(* CoDeSys 2.3 project: cy-01-wg-028.pro *)
(* Title: cy-001-wg (Albino Biblioteca E02) *)
(* Author: Andrea Ravasio *)
(* Libraries: Standard.lib 2.12.10 14:48:34, Util.lib 26.9.14 10:12:46, Visual.lib 2.12.10 14:48:34, LON_01.lib 28.9.12 14:05:10, WagoLibIdent.lib 25.2.13 11:12:16, WagoLibMBX_01.lib 20.3.12 16:32:40, WagoLibStatus.lib 2.12.10 14:48:32, SysLibFile.lib 2.12.10 14:48:34, SysLibRtc.lib 2.12.10 14:48:32, SysLibSockets.lib 10.2.11 09:20:54, SysLibEvent.lib 2.12.10 14:48:34, SysLibPlcCtrl.lib 2.12.10 14:48:32, SysLibCallback.lib 2.12.10 14:48:32 *)

(* PLC configuration (modules and I/O channels)
0750-1506 8DI / 8DO 24V DC 0.5A [Type_34_8_Channels] node 0, in %IB36 out %QB28 {INTTypePAAssignment = PLC; INTTypeModule = plugged}
  CIR09_AL AT %IX18.0 [BOOLOnX_I] Ch_1 Digital input
  CIR09_EN AT %QX14.0 [BOOLOnX_Q] Ch_1 Digital output
  CIR09_ST AT %IX18.1 [BOOLOnX_I] Ch_2 Digital input
  CIR08_EN AT %QX14.1 [BOOLOnX_Q] Ch_2 Digital output
  CIR02_ST AT %IX18.2 [BOOLOnX_I] Ch_3 Digital input
  CIR01_EN AT %QX14.2 [BOOLOnX_Q] Ch_3 Digital output
  CIR02_AL AT %IX18.3 [BOOLOnX_I] Ch_4 Digital input
  CIR01_ECO AT %QX14.3 [BOOLOnX_Q] Ch_4 Digital output
  CIR03_ST AT %IX18.4 [BOOLOnX_I] Ch_5 Digital input
  CIR07_EN AT %QX14.4 [BOOLOnX_Q] Ch_5 Digital output
  CIR03_AL AT %IX18.5 [BOOLOnX_I] Ch_6 Digital input
  CIR06_EN AT %QX14.5 [BOOLOnX_Q] Ch_6 Digital output
  CIR04_ST AT %IX18.6 [BOOLOnX_I] Ch_7 Digital input
  CIR05_EN AT %QX14.6 [BOOLOnX_Q] Ch_7 Digital output
  CIR04_AL AT %IX18.7 [BOOLOnX_I] Ch_8 Digital input
  CIR04_EN AT %QX14.7 [BOOLOnX_Q] Ch_8 Digital output
0750-1506 8DI / 8DO 24V DC 0.5A [Type_34_8_Channels] node 1, in %IB36 out %QB28 {INTTypePAAssignment = PLC; INTTypeModule = plugged}
  CIR05_ST AT %IX18.8 [BOOLOnX_I] Ch_1 Digital input
  CIR03_EN AT %QX14.8 [BOOLOnX_Q] Ch_1 Digital output
  CIR05_AL AT %IX18.9 [BOOLOnX_I] Ch_2 Digital input
  CIR02_EN AT %QX14.9 [BOOLOnX_Q] Ch_2 Digital output
  CIR06_ST AT %IX18.10 [BOOLOnX_I] Ch_3 Digital input
  AT %QX14.10 [BOOLOnX_Q] Ch_3 Digital output
  CIR06_AL AT %IX18.11 [BOOLOnX_I] Ch_4 Digital input
  AT %QX14.11 [BOOLOnX_Q] Ch_4 Digital output
  CIR07_ST AT %IX18.12 [BOOLOnX_I] Ch_5 Digital input
  AT %QX14.12 [BOOLOnX_Q] Ch_5 Digital output
  CIR07_AL AT %IX18.13 [BOOLOnX_I] Ch_6 Digital input
  AT %QX14.13 [BOOLOnX_Q] Ch_6 Digital output
  CIR01_ST AT %IX18.14 [BOOLOnX_I] Ch_7 Digital input
  AT %QX14.14 [BOOLOnX_Q] Ch_7 Digital output
  CIR01_AL AT %IX18.15 [BOOLOnX_I] Ch_8 Digital input
  AT %QX14.15 [BOOLOnX_Q] Ch_8 Digital output
0750-1506 8DI / 8DO 24V DC 0.5A [Type_34_8_Channels] node 2, in %IB37 out %QB29 {INTTypePAAssignment = PLC; INTTypeModule = plugged}
  CIR08_ST AT %IX19.0 [BOOLOnX_I] Ch_1 Digital input
  AT %QX15.0 [BOOLOnX_Q] Ch_1 Digital output
  CIR08_AL AT %IX19.1 [BOOLOnX_I] Ch_2 Digital input
  AT %QX15.1 [BOOLOnX_Q] Ch_2 Digital output
  ALARM_PM AT %IX19.2 [BOOLOnX_I] Ch_3 Digital input
  AT %QX15.2 [BOOLOnX_Q] Ch_3 Digital output
  ALARM_TB AT %IX19.3 [BOOLOnX_I] Ch_4 Digital input
  AT %QX15.3 [BOOLOnX_Q] Ch_4 Digital output
  ALARM_PB AT %IX19.4 [BOOLOnX_I] Ch_5 Digital input
  AT %QX15.4 [BOOLOnX_Q] Ch_5 Digital output
  CTL01_ST AT %IX19.5 [BOOLOnX_I] Ch_6 Digital input
  AT %QX15.5 [BOOLOnX_Q] Ch_6 Digital output
  AT %IX19.6 [BOOLOnX_I] Ch_7 Digital input
  AT %QX15.6 [BOOLOnX_Q] Ch_7 Digital output
  AT %IX19.7 [BOOLOnX_I] Ch_8 Digital input
  AT %QX15.7 [BOOLOnX_Q] Ch_8 Digital output
0750-1506 8DI / 8DO 24V DC 0.5A [Type_34_8_Channels] node 3, in %IB38 out %QB30 {INTTypePAAssignment = PLC; INTTypeModule = plugged}
  CIR01_TERM AT %IX19.8 [BOOLOnX_I] Ch_1 Digital input
  AT %QX15.8 [BOOLOnX_Q] Ch_1 Digital output
  CIR07_TERM AT %IX19.9 [BOOLOnX_I] Ch_2 Digital input
  AT %QX15.9 [BOOLOnX_Q] Ch_2 Digital output
  CIR05_TERM AT %IX19.10 [BOOLOnX_I] Ch_3 Digital input
  AT %QX15.10 [BOOLOnX_Q] Ch_3 Digital output
  CIR04_TERM AT %IX19.11 [BOOLOnX_I] Ch_4 Digital input
  AT %QX15.11 [BOOLOnX_Q] Ch_4 Digital output
  AT %IX19.12 [BOOLOnX_I] Ch_5 Digital input
  AT %QX15.12 [BOOLOnX_Q] Ch_5 Digital output
  AT %IX19.13 [BOOLOnX_I] Ch_6 Digital input
  AT %QX15.13 [BOOLOnX_Q] Ch_6 Digital output
  AT %IX19.14 [BOOLOnX_I] Ch_7 Digital input
  AT %QX15.14 [BOOLOnX_Q] Ch_7 Digital output
  AT %IX19.15 [BOOLOnX_I] Ch_8 Digital input
  AT %QX15.15 [BOOLOnX_Q] Ch_8 Digital output
0750-1506 8DI / 8DO 24V DC 0.5A [Type_34_8_Channels] node 4, in %IB39 out %QB31 {INTTypePAAssignment = PLC; INTTypeModule = plugged}
  KEY_CT_ST AT %IX20.0 [BOOLOnX_I] Ch_1 Digital input
  KEY_CT_EN AT %QX16.0 [BOOLOnX_Q] Ch_1 Digital output
  GZB_ST AT %IX20.1 [BOOLOnX_I] Ch_2 Digital input
  GZB_CTRL AT %QX16.1 [BOOLOnX_Q] Ch_2 Digital output
  VPN_ST1 AT %IX20.2 [BOOLOnX_I] Ch_3 Digital input
  VPN_DIS AT %QX16.2 [BOOLOnX_Q] Ch_3 Digital output
  VPN_ST2 AT %IX20.3 [BOOLOnX_I] Ch_4 Digital input
  VPN_CTRL1 AT %QX16.3 [BOOLOnX_Q] Ch_4 Digital output
  KEY_QE_ST AT %IX20.4 [BOOLOnX_I] Ch_5 Digital input
  VPN_CTRL2 AT %QX16.4 [BOOLOnX_Q] Ch_5 Digital output
  KEY_SCT_ST AT %IX20.5 [BOOLOnX_I] Ch_6 Digital input
  AT %QX16.5 [BOOLOnX_Q] Ch_6 Digital output
  AT %IX20.6 [BOOLOnX_I] Ch_7 Digital input
  TEST1 AT %QX16.6 [BOOLOnX_Q] Ch_7 Digital output
  AT %IX20.7 [BOOLOnX_I] Ch_8 Digital input
  TEST2 AT %QX16.7 [BOOLOnX_Q] Ch_8 Digital output
0750-0464#04 2/4 AI RTD / ADJ./ HA [Type_44_4_Channels] node 5, in %IB36 out %QB24 {INTTypePAAssignment = PLC; INTTypeModule = plugged}
  T_S01 AT %IW0 [INTOnW_I] Ch_1 signed Input value
  T_S05 AT %IW1 [INTOnW_I] Ch_2 signed Input value
  T_S03 AT %IW2 [INTOnW_I] Ch_3 signed Input value
  T_S04 AT %IW3 [INTOnW_I] Ch_4 signed Input value
0753-0648 LON-FTT [Type_55_1_Channels] node 6, in %IB36 out %QB24 {INTTypePAAssignment = PLC; INTTypeModule = plugged; DataStream = 1F8B0800000000000400ED5D796FDBC892FF7F81FD0E5C01FB9001AC5897E5631C3F2812150BA3C34349F6044920D0624BE68422F578D8F17EFAADEA2629526C5E3AE2D823609091C966755577F5AF8E2E362FFFFD63A1098FC4B45443FF5028BF2F1504A24F0D45D5E71F0A8E3D2B96EB857F5FFDF77F5D760DBDA3DBC49C; DataStream = C95322C043BA75F1C3523F141E6C7B79717CFCF4F4F4FEA9FADE30E7C79552A97CFC57AF3B9C3E90855C5475CB96F52929F84F29E94F15841BD3989BF2A2038DCF4B17A5D2C529FC7B72512A5F94EA17A51AFC28087FA9B3BEBC201F0A0DED5ED58D8958AA148421D1662D63EA2C886ECB3688D53416F81B5A298AF06C38A6; DataStream = 306557840762025B7DE29886DE56CDC5936C925B7F2CCE690743F991DCC8F6C38742F3E2EBD2B9BFD7D4A9F1B5A12B2691BFDEA9CBAF7F75DA05A167288E46FACEE29E98F06801464C1070CC7AB2F97D70FF3799DA16BDB67ED5BD08974764B1D4649B7414604D9DA9C4F4EFC15D1C8E8E72552A09BCFF2E8FDDFB81278653; DataStream = 6349AEE016FB11B8F30779C6EBF8BFC0D58EAE901F57E5CB63F6C3E7EB3881319F699C86AB61FB66A41B0A6192AD1EA437FD47B84DC34D06A63A577559E3360DDDF41FE9585D63FA9D2857B6E91090C1FB33D0A027EB8A6C1BE6B3DF667525D06CB044A591B5AB99AC59B4997FC56FD52338D16CBA7128437FFBAD448DA09A; DataStream = 350D07740D16CB85AE6A1F0AD87941380E0C08B19F0CF3FBAD6CAAF2BD46ACE0A4ACDD0BDC4AD398CDB42659737CED39AFACAB4F4085F066588752F588A34BFDDBD1C4B8FF7B6292FF38C48AD3A69546E98FAAE4358D3609294DB029579B3269540EADCAAE5951ED2AC768176D994DC31851551F125D19A90B3AB5C13FC3ED; DataStream = E41FA176813FD7DB49644AD44712681ABCB226FC8DA91AA66A3FAF84F7AF845A0E89F9A84EC9E81934AF31FDAE1B4F1A51E644016D0CDC093DD2524D400618C8AB8EBE7460525717C22C83599BA9539C9BABBEA10313C12BA1A64D439FA973C7A4060456C99298B64AACF541ED587E576BCAB27E3DF4D8C7679B0CD5FF2357; DataStream = D5CB63FF7760D51FC72FFB5F1611AA498850DD2522803B613B56064030866ECB543CF05BFEF2705039C04176381838F6EBC283FA9BC183D3243C38DD191ECC548DA08B90C53D68435B099BA6BB077ED31DE281AFE8E980E091CC800727073C78BBEE41B9F276F0A0968407B59DE241760701D7399AFE2C2EC2AAED2F0F0AF5; DataStream = 0328BC6127A172FA6650E13C92866223C4A286D24E5161696481046AFA6F8C2C41C3AAE92F0F08A7074078BB5E42DEA021726795714C65F9F29897BDDE2CA59D9CA02E966332D4C59C296ABA286F55D376644D9839FA94AD16E15E83415DCF3CE74A2327ACD5431E391BFEFF7A7964689E358F1CA59DC110F8DAB0434B9027; DataStream = 8114A765B4E5C11408BF9A6FE88B77C828B3117AB98C32B4CE98518E503E00C3DB028697F71173E2C2DBC92C9F256592CE769649B241B570F92E9659700115714832BA0C41D20760785BC0F0FA3C86B7934D3A3B4B4286B35D2183ACC9E6220B283458C32C90E0D23CA0C1DB428357E72654CE0F68B04F34C8EC231C00E14D; DataStream = 02C2EB730FDE1222246514CE769651C0989F64CA336ACF43D6360B22B8640F88F0B610E1F5B9086F060FCAA5241781DEDD0D223C3CCAD3C9C25032A142EBFA6E02939C3D9D10A07E0087B7050EAFCF5D28BF217438494487939D651AE1CA24539611A1A131B5B161C64CA34BFA800B6F0B170E4EC30116C2B000DEC28DA1EA; DataStream = 5977200EB8F02671E1F5F90B0760D83F301CFC857F3A2E1CFC85972B634A4285F39D8182F5A4DAD3872CA0D06CB71014441D472963EAD1257E8085B7050B0777E1800B215CF874C085032E1CDC85C39E843748619FA1479B1FF624FED1E0F0FA9C86C39EC41E730C080D8704C33F1D140E1EC3011322EEC26143E21F8F0BAF; DataStream = CF593800C3FE81E1E02FFCD371E1CDFB0BBB3E6463ED9A7575F93F5F9AADC6A8F1E532DB11DE974DD99635637E7589C7D6081D0BFE67139328785CB5D0829BAB93AF6B48039BE1147E28E0BFF0B7612E64DB6F54C7363DF96FC30C3C5710FCA3B2DDF3BB29194B78F7E3ACFEDB5710E10E86C4FA8A14ADAFC351A3DF6A48AD; DataStream = F7A3CF37ECC06F3CED3B06070B824466C0AF3E2589ADE89B98F86E25F053392E578F2BA57245289F5D544A17E54AE16A1DAD292BDCABC247D9724760082B756A7FA97F2B08740983F8058182E787C269B520202C7D28D08175CF82806B8F367B18710C241427C391346E8EFCA3CD6134D5297B3274966141402D43F60BC258; DataStream = 57A1B37F69F6EF1DFD51D65445B06C132616BAB10CC79C927FCDEDDFF94205D81775672178E491BB898D73F7435D380B2A0A800CFB5D2C7BC248F17288FD718F27852FFA509DEBAE62B9A27892CC024324E8F0945510903BC216833BA427088A29328D758BF6023A3587B9B0F070FA393B7C1DFE1A4EF1051AFAC74ACE9393; DataStream = EA89271EED8927DCB83FEC7CEA8BAD4977D0FF541006B399456C4A282AB0CA886067A41110B71212D76DB56F895C4817F0ED62C3E14E5C8C6C55FE645272139F5CBC940B55D3548B4C0D5DB132C90933FDA5BA5A4BFE026A81568095474D106445011DB7F8627406FD15FB273CF615D4729F0663F8C463D8C321BF938CEBBF; DataStream = B2E2B9E2F1DC6024041B1F03E0B5CDE7A4B59FC834B2637BDC563D6E793D64D5A5E1838114B32853B51AC0816A35221F3502093A35BC1E4869023222114DF2E1E1AC78AFDA82E3322F00E2310769BF2B273CC06A4E64A86F840CE57A9CA8EB8E0375A336B14FAE6971EE756217F10B0A496B2A937E5A7AFC52B238FDEC414B; DataStream = CB01252DBF261DFDA8DAFEE4AC09E4829FB190559DC7FEC7CEA89DA26F8AFB703CDBFE44B1A6B9AD92702A5011E09F804D74053A0D0A5439F544EA83326C28904E1F8D1787EA994E23AD3C42D42242D47C216A4121026615F05698629374514EF99694DA840459A818823113B0A94AB219D18D251A99B26EC934E4A1CE8299; DataStream = 2ED71977A1FC98B88FC78B461BC0E8C164E505F31CA050393909C35D1E1038E7229D4B265E32D622A8825B00F7E9B7E052622C7C320D67B93564CF97F1903D0FF5B03580A5A17058A536C2DE7BC3D088ACEF03B6EA2B15823E37E4DFA28F66006136F4ACF93FDE74303EC6BA6341DB994A346543511C4A224994B448FA604A; DataStream = 0EA62404C05B5B9239A3B29D4AF24DCB2606673397DB0578C77EC03D81298BD00D2EE2C40D4EB9C48D7881E4C448449FFC98BF896C5E8E3BAF54DCBCD01288E5906A0BC7A1F62DB842BD8C642D94916467506E9A90F49E76E3D7D3DDE724590FA19464B9CCCD490E6325894B49AEB84FCC48B266F109C9FAFE93107D1FB991; DataStream = A398BC57F6D424330413633671C9C5A7225C83B46F01874423539B5A782D394ACF909DB45C6213466C671958CC4C2664F936CD46CA8AE973B6B3ACBE0B013189D4A9A92E6D836B9033050E4A80C4AE396F98A6FCFCA55CFF86EADE6633343304192F0B846D95AE3C5EDC6AB1E82301BCF69FE209D890A4C6E714F928F43002; DataStream = 2E22D43DF1181FC05AB92E4C1F64131C1C62664812D3D5D1840732DA1E04D300CA55CE22C2AD0F09672ED992695E37A495C015AEADF525FE523EF9B6B666E2D09125BB1AC366A7B31A8ACD8D16EDE74F4756323A63E5DA69EDAC5AAF9DA6C566EE30FC396EB402C3C045464E8CB6267DCD37D2CF762E0F7A43641CA5A52DC3; DataStream = 8058C9133A675EB33B7544524133F3764860FBE67CB7F0C3D08785CE42A715833E5CF0F11FDA147C58203D51154FB628F6D405A67DFB8D7162C5DFD6B1F725FC12C19A6CD9F49F14DCD4D7464223FADC7ED83E0470E5F7C8C50F80D817CAB5F3D259B1ECA557BC677EB94C291624EC2655BAFB382E7DD321562AAE839977FF; DataStream = 214F84BE05CC96035B7CE5550DCA5935182211E1119CE364DF2F26E4A3870C72362BD185561F5505BFA1830B96AED31DE48C19BB48B1149F3A8AF20A0F94769333884F4CA6F05BCEC96F793FFC56B2F25BC9C96F653FFC56B3F25BCDC96F753FFCD6B2F25BCBC96F6D3FFC9E64E5F72427BF27FBE1B79E95DF7A4E7EEBFBE1; DataStream = F7342BBFA739F93DDD21BFD9383C4B4FD6735D1B78F6EC85C1F77C73D6CF5F1887CB09862E8DF7F29E8C5E66502E2758BD54E6F7640133237439C104A632BF27739819AECB09F63095F93DD9C6CCD85D4E308EA9CCEFC9506606F27282A54C653EB3D5DC59D59F1711F859182C8817E8D786368807569F2AF2B8F737809E89; DataStream = 6C1E090B43B71F8E04457E3E121E0C07AFA8BA63932381150467CC9A66CF9C554B58E5CFD91CFA4C647EC413CCA145C57CA68F25A5032B4189F3A40373C5AF9E183D1CD03CF12B37285F302AF1BA471BEC4998EA2A5126738BA1E344E146E28A9C58F100B7F72446C50FAAAF41B1F3C851E3C9F14089C40B82F7F724C9C9B9; DataStream = AF5D74716E5D23BB70C924E8176DB17779860C6472C8C32D1C72B12A29871578BD619BFC4D204F5E5EEDD89FF95B3FF42B319B6FD9D3CFC6F8C0B5978C79D770EB3F7224CCBD6712F2E5518134FFA197CD91C709BCE51AF2C4CB97204781B7CE8F6FB84FC55E3D8CD9F6C8F376844109B1ED8FD80D2BD628F3DE3DAD27A1EA; DataStream = 3FC1ADB0503949B512F218AAE1C566C76CBFB19A92C4BAB5557F499BA8B2DF4D7C85C9695611976EA1D244238F44CB5235E39736D127D225E596B185BB4D927619EA2E5EE2B39FF4921F0245FF364F3D0D77438BEAE1C4362688B3497AABAE3A15A6B26321D8BAB09C2A2FC3D91AC5D95B4CB1C7806C8D07B2B76CEF2C7547; DataStream = 92BF8DE3EEBCADED80FB505BFB2950CB9539C7560E1768A964B44C262114FBB9B0CA8298E4B8254E3BB988CA89625E41E852E682EAEB8C5DCA5CD87C85C10BBF78E895462FFC12A0571CBE54F87BF0B9E2975DA3D9F9796086FC57C1F354347103FF4590D6CEDE3E0F9A58E6FF69EA023CEC1C8636F0580673CB2FD7629EA3; DataStream = 4BE3658D6EC228E4D0CB04FF9892DECE006F117287CB795DE7F3DC37BFB4D67269586A5C7C9AA5481E9E8F44A94B3CFD8C98475E3DCFFE8B2325222BC777E07BA340B4F3D45249CE2B464F93A59D9211F535955657E3D4ADDE53DCFF3117BE90196AB5C238C3CDCB81C0B1555A3EC8ACDEAB5AD584EE5C277D47CA0DB4373F; DataStream = 4A0662E749E03496D071129DD6914FF9174A18FCC42C814B9877164EA5C60DA1D327241C42738D74B8DBA410DA0875171F4263A4BAA52206368F2AABDDA3F3EA9AE41B27245113C3AF10D5838AE8BE7833D3E4797633F766B431B558C3CDD9163B2D3A44E91B915CC55319153EEF3BD84A2D6713C253E71D48B25A433FBF94; DataStream = A3A55A4844D9460EC5A5F122E51C03C72E1AB322F5CAAC6DA4301C1B5F3063845EA4B863B0247A71AA9A5347DD4AAF0CA03371E9BC48A1873B27163B39710793E2527A91C28F1E993EC8BA0A1D1767B2A36D35330B9FD684D27A9162903621CABD3CFD0EE2A89A636E353F3397D6C4A5F593CAFE068FC42C9AB23ECFCA3C37; DataStream = 243780CA845279114B3206BBBA03291C24B34F31522C8888EFAE9AB9D7075716E2D3DAE7FA48B12863FACDA0A26D141744B6B22F9098D94162B8D3E2127B11CBD234160B47778F3AB0722E7CAE5C53A0B887459FDDC6B4A16FA2808DD166453BBB23C61506E59820A589BD373F2CADBCD093A3A8EAC5257288870F6D21932F; DataStream = CE44D5271EC117B137EC24E22298F26DE4D1289509FFF0CE7DD8989EAC3B80695343B74D43CBC83A3727B3A094262EA5178A5A96E093B1ADFB2D240155F26A727EBEA16132A0D13655252B78C589E19179110B2391A561DAC5856C7DDF460C939299209917B12A1E47AA3E2FE2D7B1B69165B9A245BFB4F52236252810DA84; DataStream = 5D0984B45EC4AAD0CD90A26ED8EAECB9A8E40BF5B952B12D104670B2DFB83FC5AA48C4E2BFEF9B69E1C03DC0E3C55223C93BA71B1CD17726044D8B5F0A897D9A8F44C9F0DA06778B2DF0FC3E4EDFDA22D1BF7A079B7E407383B4AAE53EB8967FA4A52E2CAB4AF6B26BB82A5B89AD365ADF218C2F357227C57B47E223CBB8AF; DataStream = 4DD0FFD223911C4DF3CAD752F56AB8CD99C2E1C3A692CE1A59AFFF883B7E2AE5B0115F50DA969E6FB7E5F92A6E7ADCDB2238C958F85239AD87CEA3A99C56CBFED6227EB105F71E68EC92FB1D8BC0A75CC283E14D7B25E9B50B8580274E2CA149344B75B26C31D25D1EFA094A3B3010672145E6CEF9F56DA3292C620E10883B; DataStream = 632CFCC1CBA429F6C9276CE9D46267DFBABA0CB40FFF25ACBE9C3092E7EE593FAB0DAEAB4B5659174AC80BEE128E4AD49626FD71B72048F2136DC386E8384C6588D4755B9535419E4E31F63209EE5D73C90D6EC4FE6434980CC57E2B03A527DCDF4D2125894DB1732B06B98C32D9D40C8B08B20EE02E3F12F7E8312ED96677; DataStream = 301427ED4E3744B192405121680BD369B6C4AE388A92AE46484BF4C84E6053A19FA431CC67EF7B025CEAAD0E0CC168207D867537F8637C13245E8B1207968D45CEA99A488D20D59314AA39A66D8D323B60EF38A0D15CF5AE07D5DB3F3730AF760F3368372D0BB1F178D3193105CBA10282198A21F8575B0411FF889069F933; DataStream = A919C6773CF2378D129B4B4A2B49B145D3344C014FE15C121DBD9658351CB2A16F373ADD64CDF6492A6B4C27732A4A52B25A878752D585556E257E2CC7FD9628DD611D559252FB2CA33EC3281CA306A68C4667B0CE7254ADC32CE34B908A40F3285C8AA34E4F1C8C47EB64EB11B2772AAC9627C1A27837250241F66388DE75; DataStream = FAADC1DD3ACDD308CDB54359FD04239768633CBA5E27791625C956333354860D3ABBC4B099F01103A8369BE2700853D6B85D53B2F314C0B827CF0620A938E09E8A00A487A2F8C7A4D3BF6D7471DB3EB0204AD139735BDF353A5CAF337C3F40AA9C0D7B4E5DEC09BD63126661BC54D087F3E7F701B4927027B8D19D5C8B0D50; DataStream = F1300C4517CF3AC99961D8B124DB83C1689D64749DB7C8BD33A7C70BE207BD50C27738CBB2CE5E53F82D86784BFC38FE14A61D85A54E80AAC358CF44BCD36F0FC2B4A3133C7CB6C087CCCFF8F0F37024F6A25D44D7E7E8C13D5B5A502DC1AD3588210A1A3916799A598CA24988AC0C2EBE0EA64B770F51CA264373D0C7AFA5; DataStream = 8514B718C543EC4921740B19BA3266334DD5B958002407ED76B7D30FB924C5A8FEB1E2502CAE55D9A4EAF8A53F18F985FC0CCB5750A0A56D50A9021B261E0C0980CE0FB2A93CC9B877C2AEC58938EEFFD11FDCF543FC4495D7B3EE8177AADC6194D738A5C8B52453FC84A512D769BA23D0378475CA4BCC2CE85C6B80240738; DataStream = 5BADCE881E0BBBBE9C759FA59C641BDD5E906E926F30326C593BF66A096821E823FAD6B4BFB2F00ED338860E5DD10A3330F696E03586F9C233E86CA2CB803671A3361A8C26C3DB26E5A99CEC5424F2C2DD205FA35F49762E12E973B745D6E857933D0CB7381AACB65B20CD264D23B22970437E20DF05BBDDED8DC0FD97C2C3; DataStream = 13858624F271A313245F49763818F90775FE9083FDEBCEA76B3EFF1CEF23A9833801421D54527C11EE00A58D7C4431A38E089F70DA9847349263A762C62475B8234C73EC6B0CEDD4918EF21D5DAA6D408275508A73343A12920C11E439FE401050AD989DE88D244608471725122E9A04BF35AC809B6E38F7E0AEBFA3F50FBF; DataStream = 65EA66247D0CE17E99170204FA000F1811C632E8F73B3CC07E47DECFDF1F81913155FDBB06810222B89560E2B0EBE1F8E636D47574D586C5C31D6EEA8A671FC591381C458631BA7863FAC93763B42FDEB445D772A8BF054BC509447F544D43C7F74D00B7D13411DD624E047B811842BBE9033FF6705910FBB7CD41EF66D26B; DataStream = FC15E220BAE8431CC8F73A3A921A588DA5636712B637E8774603891AE290DDE3842361617D9B0AD348CC38234FFB6874FA387BA214F2F62A9C1C057ED15790974BCD73BB62034AA4DD18C1BF10FC0DC2F17A94F501449426A3953A2A517A513E193DF00169A2228DE25D43EA77FAA148A35AC916A29DB9215AE41DF99C19A2; DataStream = 9B2CF9CFAEF18445346CA52CD7DEB1E7D2EC8AB76277121D6FFF16D74404EF26797D7E3BAE3108DE4DF2D7AEC1B46C245635D94FEBAA33220CE5190162D42E504B6609EF3E369A7838B07F4841850B9E376B9E48D426DCB0EF683F67EAA41AD74925D95DA344870163C0EC71847E2D8E7E35D95FA3F447CCA01DB7696DE0BB; DataStream = 966A2D35F9F9B7682F2771BDD4929D36DACB0DC013E5FE48A0DB124DCC9C4D014F4408099608C771C2D5E3BAAD27BB72B49BB819398B237A96ECC6C5F12E8DFA474C07E057D220964BB10A574A71F468DF94BCC6B0C05B2EBC6E6247AD5CE7F87CA95087EC50AC8BBCCC9413EBA43F33609D486B32DD17A7E8E6874916C623; DataStream = 5CF18B82F8940752AFD1E564C5AD00BD98675B9D61E363576C25A31E2B0CF238F3DE34E2121CDFB41A23DC596F8CC6C36414BC212626997CB25EA9610CE5A1D86D5347281903DD5C9E1C3AE22989D546B721F59261CF95DF7D8F0A8F0A62C54D5CB29278339046E0610CFF48C6B9815732963843835BB0FE9D96988C6921DD; DataStream = 89A124F671AA93514B72358E4D498AE249BD5B2E7B51546AD250358BFE34BB6243E2A84F14944234DDF2BF04929169E6608D3B8A4C77683591EA9D8EC5A54C69C2FA1B75DA9FDDE16D717086B72A37EB83BB5C399B4C212499D17C13D67A0A7EAD27B7AB5EA33FC634E8480AC76DD14516ED00A18A565624752089BD01ACB8; DataStream = 48079C3D27D641A05A0D2B54685A8F893153E78E0BD64BE694D0EF3072BBBD91069FA44678F2A3CB91E913ADC12A7A3558B4264D78172ECCE2DA185FCF24712886B73E38ABF507993A409D75E66F3B8084890B384A3ABA8099140081B2A019F3444EBB8390FFCF8925BB860C31EB833F0FAB542FEE300E9B3723BCC1BE3916; DataStream = D35577D068712780B36BE5E8B4B3A9639AE05D68B8332A2BD097DBFB7BA1330B71F3245BC283ACB1D80FF55B7B3E8206AA253CA91AC6B4165874C17474B6776B1A0BF638BEB68FA9FBD5F3EFE3467CDCE731CF8944AF814E0AF7239FB3A55B35171E5B5A9A84665FC6EFBC33AD001F0B4605D3FE78232856F0512ADA13C47F; DataStream = 4400DB942ED675A33BE2CAC533FDC097992CDA6A68EFC95CA5A31D3BA060BF1B12BFF3288E8D75CDD3C0B8BEE36C7B3F4EF12A1C3463CBD1A21DE9E4878D4B87BABAC6D2F308DFE1268F5BF487BEEF11AC008B961FC2DD23F680708F6F031C09C49EBEFF0D57739A3EAC4FFEC201FFF69E08FFFA8F63D8BFAB8A46D82FDC31; DataStream = 60BFD8BCBA57714B683A254B9B29BDAB25478281A98027D562DA803A0334D5B96E98A012A16E4D623BA66E21250E7D57236736262AE818D12F92CE42DDC5796B23F1863BFCB58CAE77CD75BDDD0A33BEC3FD18E77063D490C1E56E3273856945D9B10D4A0061043FC3A6CF09EE9DDB4F84E8A1FC0FE6EFB8A68676DA188F06; DataStream = 51742032AD9830748D5B68449FBC161BA3643FBCB1E2A2E842F114D861299F27ACA9E6D79150F23DA9FF697227F5C2354C9CDA2BC3D052796D0E06DD643F9CCBABAECE1F208273CC79C2AC753E5D03408CA54F62B257CEED01F3AA5383EF8150F298455DE79EE30CAC1403B7385DB7868D8B632F1D3B5E0106ED768AAFEEC7; DataStream = CFF7040962CCC34FBD527AEB214FD4E68BB078E6E0413C632D84CD4A4ADED19F4B67B1E4BA2B94B2D813A54F11B5E36C0FA9FE28B0A422019099C960AD013CB06887EBBBD22EDA8DFE64D0EF7E4E71E55D957B52ED079A9DC614BFC13A75CD777C0F92189D508E6FDF9992E242FE8EDDB00AD2187A9DA698E2C2BBF5AD74B0; DataStream = 53C9F51A7F451736C76387B13516A0BF8814C7381EC964C5E6A03FE87D4E71D35BE4C159A88A1F6224D36C89D7E3DE5A055074D5350178EFCD0CE49A8D6EE7A30411768ADFBDD2DE69BAD8546323B3CD59633E51585B60E83250058BD548DBCCF1A794B19030E7111EF9A9BAC9F56D93FAC8F156C16F90E83C33E81C24D3F2; DataStream = EF475CD9B03D3E0E97401F63A5DED525ADD7EB58F03F7008DCDAEB16041AB7C4B4A0216ACB7BA086CD5851777B0951419BD611F96D4EB0494FFEDB30038F01C3B2FD00BA75F1D5E59C52B184773FCEEABF7DED1AFA9D617EB7BED202EDAF58A3D36A48ADF7ED1BB706AD03CC944A02EF3F9095CC805D88AF125BE1071C86F8; DataStream = 09065C9EC7E5EA71A554AE08E5B38B4AE902D62B48EFE8D4D79335E8917EEE9973CDF75EBC5A77FC4E9E30F0833A559FAA4B598B39B5600802E127EFDCF691027C18FC1E785C32568DB2F70A081E98C53E6A1DE874FD20A5684FFAA32A7977715003876345EBFE53BA5D3F502B3EBDA33F1ADEC7C5839D56B99D863BF15FE6; DataStream = A14A982C193601E9429D9C66E9A41EEA24510E6C81B2843BA965E8E434D4C9EA4CBC58516E8CB5F172576C44F978D756ABF7B8891B99C6FCEADB37F8A38BEF42C0329EC95372F5FF61272651A0F00000; DataStream = .; DataStream = .; DataStream = .; DataStream = .; DataStream = .; DataStream = .; DataStream = .; DataStream = .; DataStream = .; DataStream = .; DataStream = .; DataStream = .; DataStream = .; DataStream = .; DataStream = .; DataStream = .; DataStream = .; DataStream = .; DataStream = .; DataStream = .; DataStream = .; DataStream = .; DataStream = .; DataStream = .; DataStream = .; DataStream = .; DataStream = .; DataStream = .; DataStream = .; DataStream = .; DataStream = .; DataStream = .; DataStream = .; DataStream = .; DataStream = .; DataStream = .; DataStream = .; DataStream = .; DataStream = .; DataStream = .; DataStream = .; DataStream = .; DataStream = .; DataStream = .; DataStream = .; DataStream = .; DataStream = .; DataStream = .; DataStream = .; DataStream = .; DataStream = .; DataStream = .; DataStream = .; DataStream = .; DataStream = .; DataStream = .; DataStream = .; DataStream = .; DataStream = .; DataStream = .; DataStream = .; DataStream = .; DataStream = .; DataStream = .; DataStream = .; DataStream = .; DataStream = .; DataStream = .; DataStream = .; DataStream = .; DataStream = .; DataStream = .; DataStream = .; DataStream = .; DataStream = .; DataStream = .; DataStream = .; DataStream = .; DataStream = .; DataStream = .; DataStream = .; DataStream = .; DataStream = .; DataStream = .; DataStream = .; DataStream = .; DataStream = .; DataStream = .; DataStream = .; DataStream = .; DataStream = .; DataStream = .; DataStream = .; DataStream = .; DataStream = .; DataStream = .; DataStream = .; DataStream = .; DataStream = .; DataStream = .; DataStream = .; DataStream = .; DataStream = .; DataStream = .; DataStream = .; DataStream = .; DataStream = .; DataStream = .; DataStream = .; DataStream = .; DataStream = .; DataStream = .; DataStream = .; DataStream = .; DataStream = .; DataStream = .; DataStream = .; DataStream = .; DataStream = .; DataStream = .; DataStream = .; DataStream = .; DataStream = .; DataStream = .; DataStream = .; DataStream = .; DataStream = .; DataStream = .; DataStream = .; DataStream = .; DataStream = .; DataStream = .; DataStream = .; DataStream = .; DataStream = .; DataStream = .; DataStream = .; DataStream = .; DataStream = .; DataStream = .; DataStream = .}
  AT %IB8 [BYTEOnB_I] First Byte of 24
  AT %QB0 [BYTEOnB_Q] First Byte of 24
0750-0478 2 AI 0-10V 16 Bit S.E. [Type_8_2_Channels] node 7, in %IB44 out %QB24 {INTTypePAAssignment = PLC; INTTypeModule = plugged}
  VRD02_ST AT %IW16 [WORDOnW_I] Ch_1 Input word
  VRD01_ST AT %IW17 [WORDOnW_I] Ch_2 Input word
0750-0556 2 AO ±10V [Type_14_2_Channels] node 8, in %IB68 out %QB48 {INTTypePAAssignment = PLC; INTTypeModule = plugged}
  VRD02_CTRL AT %QW12 [WORDOnW_Q] Ch_1 Analog output
  VRD01_CTRL AT %QW13 [WORDOnW_Q] Ch_2 Analog output
Fieldbus variables [FB_VARS] node 1, in %IB0 out %QB0
Flag variables [FLAG_VARS] node 2, in %IB0 out %QB0
Modbus-Master [MB_MASTER] node 3, in %IB0 out %QB0
*)

(* Global variable list: Global_Constants *)
VAR_GLOBAL CONSTANT

	Plant_NAME			: STRING :='cySN:1 cyVER:28 - Albino Biblioteca E02';
	Plant_SN			: DWORD  :=1;		(* S/N Impianto di telecontrollo *)
	Plant_SW_VER		: WORD   :=28;		(* Versione SW installata *)

	(* Parameters *)
	Plant_DefaultTAmb	: INT	:=100;		(* [.1°C] Temperatura ambiente di default in caso di rottura sonda *)
	Plant_MaxRunTAmb	: INT   :=250; 		(* [.1°C] Temperatura ambiente massima funzionamento impianto *)
	Plant_AntiFreezeTAmb: INT   :=-40;		(* [.1°C] Antifreeze temperature, start circulators *)
	Plant_VRD_TAlarm	: INT   :=450; 		(* [.1°C] Temperatura di allarme VRD, blocco *)
	Plant_VRD_TMax		: INT   :=430; 		(* [.1°C] Setpoint massimo per uscita VRD *)
	Plant_VRD_TDefault	: INT	:=300;		(* [.1°C] Temperatura di default in caso di errore climatica *)
	Plant_CirOffDelay	: TIME	:=T#15m;	(* (Def.T#15m) Ritardo spegnimento pompe per ricircolo caldaia *)
	Plant_MaxWaterLoss	: WORD  :=2;		(* [lt/h] Massima perdita del circuito *)

	(* Filesystem *)
	FilesPath  			: STRING :='S:\';

	(* TCP Logger *)
	Logger_SERVER		: STRING:='';
	Logger_IP			: STRING:='192.168.100.3';
	Logger_PORT			: WORD  :=80;
	Logger_GETSTART		: STRING:='GET /cygmsrv/hsgm.ashx?';
	Logger_GETEND		: STRING:='$R$N$R$N';
	Logger_CHECK		: STRING:='True';
	Logger_CRLF			: STRING:='$R$N';
	Logger_DataFile		: STRING:='S:\LOG.DAT';
	Logger_DataFileOld	: STRING:='S:\LOG.BCK';
	Logger_IndexFile	: STRING:='S:\LOG.IDX';
	Logger_ConnRetries	: BYTE:=5;
	Logger_RecoverMsgs	: BYTE:=100;

	(* TCP Remote *)
	Remote_PORT			: WORD  :=10;
	Remote_WELCOME		: STRING:='Connected$R$N';
	Remote_OK			: STRING:='OK$R$N';
	Remote_ERROR		: STRING:='ERROR$R$N';

	(* TCP Sockets *)
	MAX_SEND_TCP_SERVER					 : DWORD:=3000;(*60000*)
	MAX_RECEIVE_TCP_SERVER				 : DWORD:=3000;
	MAX_RECEIVE_TCP_SERVER_SOCKET	 	 : DWORD:=1500;
	MAX_SEND_TCP_CLIENT					 : DWORD:=3000;(*15000*)
	MAX_RECEIVE_TCP_CLIENT				 : DWORD:=1500;
	MAX_RECEIVE_TCP_CLIENT_SOCKET		 : DWORD:=1500;
	MAX_RECEIVE_UDP_SERVER				 : INT  :=1472;
	MAX_RECEIVE_UDP_CLIENT				 : INT  :=1472;
	CONNECT_WATCHDOG_TIME				 : TIME :=t#10s;

	(* VISU COLORS *)
	COLOR_RED 		: DWORD:=16#2020F0;
	COLOR_YELLOW	: DWORD:=16#20F0F0;
	COLOR_GREEN		: DWORD:=16#20F020;
	COLOR_GREEN_OFF : DWORD:=16#006000;
	COLOR_LBLUE		: DWORD:=16#F0F080;

END_VAR

(* Global variable list: Global_Retain *)
VAR_GLOBAL RETAIN PERSISTENT
	CAL01_Clima : typ_Clima;
	VRD01_Clima : typ_Clima;
	VRD02_Clima : typ_Clima;
	CTL01_Count : DWORD;

	Mode_Manual : BOOL := FALSE;
END_VAR

(* Global variable list: Global_Variables *)
VAR_GLOBAL

	SYS    : typ_SYS;

	TPV01  : obj_TPV	:= ( ID:=1 ); 							   (* T_S01 *)
	TPV02  : obj_TPV	:= ( ID:=2 , IN_WMIN:=50 , IN_WMAX:=800 ); (* T_S02 - CAL01 - T_Send *)
	TPV03  : obj_TPV	:= ( ID:=3 , IN_WMIN:=50 , IN_WMAX:=800 ); (* T_S03 *)
	TPV04  : obj_TPV	:= ( ID:=4 , IN_WMIN:=50 , IN_WMAX:=800 ); (* T_S04 *)
	TPV05  : obj_TPV	:= ( ID:=5 , IN_WMIN:=50 , IN_WMAX:=800 ); (* T_S05 *)
	T_AMB  : INT; (* From T_S01 *)

	CAL01  : obj_CAL_VT100GC1B := ( ID:=1 );

	CIR01  : obj_CIR := ( ID:=1 , CIR_AUTO:=TRUE );
	CIR02  : obj_CIR := ( ID:=2 , CIR_AUTO:=TRUE );
	CIR03  : obj_CIR := ( ID:=3 , CIR_AUTO:=TRUE );
	CIR04  : obj_CIR := ( ID:=4 , CIR_AUTO:=TRUE );
	CIR05  : obj_CIR := ( ID:=5 , CIR_AUTO:=TRUE );
	CIR06  : obj_CIR := ( ID:=6 , CIR_AUTO:=TRUE );
	CIR07  : obj_CIR := ( ID:=7 , CIR_AUTO:=TRUE );
	CIR08  : obj_CIR := ( ID:=8 , CIR_AUTO:=TRUE );
	CIR09  : obj_CIR := ( ID:=9 , CIR_AUTO:=TRUE );

	VRD01  : obj_VRD := ( ID:=1 );
	VRD02  : obj_VRD := ( ID:=2 );

	CRON01 : obj_CRON := ( ID:=1 );
	CRON02 : obj_CRON := ( ID:=2 );
	CRON03 : obj_CRON := ( ID:=3 );
	CRON04 : obj_CRON := ( ID:=4 );
	CRON05 : obj_CRON := ( ID:=5 );
	CRON06 : obj_CRON := ( ID:=6 );
	CRON07 : obj_CRON := ( ID:=7 );
	CRON08 : obj_CRON := ( ID:=8 );
	CRON09 : obj_CRON := ( ID:=9 );
	CronEd : obj_CRON_EDITOR;

	CTL01  : obj_CTL := ( ID:=1 );

	Logger : typ_Logger;

END_VAR

(* Global variable list: LON/Module_1/InterfaceBlock_Module_1 *)
VAR_GLOBAL CONSTANT
(******************************************)
(* Automatic generated code, do not edit! *)
(******************************************)
	abSignature_Module_1 : ARRAY[0..15] OF BYTE := 16#DA,16#82,16#20,16#30,16#AE,16#3B,16#9C,16#43,16#85,16#6E,16#0F,16#57,16#0A,16#4B,16#E9,16#A2;
	wConfigSize_Module_1 : WORD := 406;
	abInterface_Module_1 : ARRAY[0..101] OF DWORD :=
		16#30A640D5, 16#2177270E, 16#6041B800, 16#06246830, 16#428B2E71, 16#64B95263, 16#FE000902, 16#2A050140, 
		16#0028C08A, 16#760610FF, 16#C5CE0103, 16#0E083060, 16#AE8EB93A, 16#EA38A9E3, 16#2CB43A56, 16#B03AA63A, 
		16#3A9E1A3C, 16#91B48ED9, 16#124ABE0E, 16#72A6C91A, 16#6102A5E9, 16#2A54A353, 16#927DEB96, 16#5AB14FCB, 
		16#A43BB6AC, 16#B26483EE, 16#FB362F48, 16#6341CAAD, 16#B66DDBB7, 16#41D2755B, 16#ACDCB268, 16#BA8509B0, 
		16#59A969ED, 16#2D5B376E, 16#0921E8CE, 16#08E2F185, 16#EED4B711, 16#D6A51B96, 16#92298CE6, 16#9BD6E800, 
		16#290A9565, 16#4DA49AC2, 16#5662494C, 16#F542D994, 16#E66C7A0B, 16#5A0509F0, 16#B3425FA9, 16#E2CA9258, 
		16#EEA4A52A, 16#812B3B15, 16#0DCB3628, 16#87F8DACA, 16#97AD54AB, 16#C01F3197, 16#454A5420, 16#304DBF5E, 
		16#25843188, 16#52053441, 16#0BB86DCB, 16#D02C521C, 16#79409EB4, 16#D1A18743, 16#A25285A8, 16#2636ACDB, 
		16#8E5E1758, 16#8930F367, 16#9EE50249, 16#538D4224, 16#865F7F47, 16#08C400A2, 16#C9FE031C, 16#B0413816, 
		16#C084920C, 16#8A838C21, 16#036D23C0, 16#B0813398, 16#38306673, 16#59E6720E, 16#F00E02FC, 16#3A02343A, 
		16#18183BF8, 16#80800700, 16#82078140, 16#07424080, 16#142E0B83, 16#C303024C, 16#2E129789, 16#71D9585C, 
		16#11C7E5A1, 16#5C3E2097, 16#A0585991, 16#41700267, 16#74191320, 16#13C476C6, 16#02C2BDD8, 16#0E140880, 
		16#48C1DA09, 16#DEE91A26, 16#B7858772, 16#AAF0EA43, 16#B245A75F, 16#000080CB;
END_VAR

(* Global variable list: LON/Module_1/Runtime_Module_1 *)
VAR_GLOBAL
(******************************************)
(* Automatic generated code, do not edit! *)
(******************************************)
	mbxModule_1 : MBX_Full;
	InDataTelegram_Module_1 : ARRAY[0..255] OF BYTE;
	OutDataTelegram_Module_1 : ARRAY[0..511] OF BYTE;

	xInitRunning_Module_1 : BOOL := FALSE;
	unLastLen_mbxModule_1 : UINT;
END_VAR

(* Data type in LON/Enumerations *)
TYPE alarm_type_t :
(
	AL_HEADER := -13,
	AL_FOOTER := -12,
	AL_DEBUG := -11,
	AL_INFO := -10,
	AL_SYSTEM_INFO := -6,
	AL_VALUE_INVALID := -5,
	AL_CONSTANT := -4,
	AL_OFFLINE := -3,
	AL_UNKNOWN := -2,
	AL_NUL := -1,
	AL_NO_CONDITION := 0,
	AL_ALM_CONDITION := 1,
	AL_TOT_SVC_ALM_1 := 2,
	AL_TOT_SVC_ALM_2 := 3,
	AL_TOT_SVC_ALM_3 := 4,
	AL_LOW_LMT_CLR_1 := 5,
	AL_LOW_LMT_CLR_2 := 6,
	AL_HIGH_LMT_CLR_1 := 7,
	AL_HIGH_LMT_CLR_2 := 8,
	AL_LOW_LMT_ALM_1 := 9,
	AL_LOW_LMT_ALM_2 := 10,
	AL_HIGH_LMT_ALM_1 := 11,
	AL_HIGH_LMT_ALM_2 := 12,
	AL_FIR_ALM := 13,
	AL_FIR_PRE_ALM := 14,
	AL_FIR_TRBL := 15,
	AL_FIR_SUPV := 16,
	AL_FIR_TEST_ALM := 17,
	AL_FIR_TEST_PRE_ALM := 18,
	AL_FIR_ENVCOMP_MAX := 19,
	AL_FIR_MONITOR_COND := 20,
	AL_FIR_MAINT_ALERT := 21,
	AL_FATAL_ERROR := 30,
	AL_ERROR := 31,
	AL_WARNING := 32
);
END_TYPE

(* Data type in Errors *)
TYPE en_Logger_ErrLev :
(
	EL_Log			:=0,
	EL_Wrn			:=1,
	EL_Alarm		:=2,
	EL_AlarmStop	:=3
);
END_TYPE

(* Data type in Errors *)
TYPE en_Logger_Status :
(
	S_Logger_UNKNOWN := 0,
	S_Logger_IDLE,
	S_Logger_WAITCONN,
	S_Logger_WAITTX,
	S_Logger_WAITRESP,
	S_Logger_ERROR
);
END_TYPE

(* Data type *)
TYPE en_SYS_Objects :
(
	EO_SYS		:=0,  (* PLC *)
	EO_VPN		:=1,  (* VPN *)
	EO_DOOR		:=2,  (* Door & access control *)

	EO_CAL		:=10, (* Caldaia *)
	EO_CIR		:=11, (* Circolatore *)
	EO_CRON		:=12, (* Crono-termostato *)
	EO_VRD		:=13, (* Valvola miscelatore pannelli *)
	EO_CTL		:=14, (* Contalitri *)
	EO_CTB		:=15, (* Contabilizzatore *)
	EO_TPV		:=16, (* Temperature probes values *)
	EO_PPV		:=17, (* Pressure probes values *)
	EO_PBV		:=18, (* Over-Pressure Alarms *)
	EO_TBV		:=19, (* Over-Temperature Alarms *)
	EO_PMV		:=20, (* Under-Pressure Alarms *)
	EO_GRU		:=21, (* Gruppo termico *)
	EO_PDC		:=22, (* Pompa di calore *)
	EO_SOL		:=23, (* Pannello solare termico *)
	EO_ESOL		:=24, (* Pannello solare fotovoltaico *)
	EO_GAS		:=25, (* Contatore GAS *)
	EO_PORT		:=26, (* Misuratore di portata *)
	EO_FPV		:=27, (* Flow probes values *)
	EO_ANZ		:=28, (* Analizzatore di rete *)
	EO_SCA		:=29, (* Signal Control Alarms *)
	EO_LUX		:=30, (* Base Illumination point *)
	EO_LUXM		:=31, (* Metered Illumination point *)
	EO_PSG		:=32, (* Sensore di passaggio *)
	EO_HVAC		:=33, (* Heating, Ventilating and Air Conditioning *)
	EO_HYGRV	:=34, (* Relative Humidity sensors value *)
	EO_COOV		:=35, (* Carbon Dioxide CO2 sensors value *)

	EO_ZGW			:=200,  (* ZigBee - Gateway *)
	EO_ZRM			:=201,	(* ZigBee - Repeater *)
	EO_ZREL			:=202,	(* ZigBee - Actuator rele *)
	EO_ZTHL			:=203,	(* ZigBee - Temperature Sensor *)

	EO_ASGW			:=250,	(* ASi - Gateway *)
	EO_ASCBI		:=251,	(* ASi - Input Board, Ciabatta *)

	EO_LON			:=1000, (* Bus - LON *)
	EO_MODBUS		:=1001, (* Bus - MODBUS *)
	EO_MBUS			:=1002, (* Bus - M-BUS *)
	EO_MODBUS_TCP	:=1003, (* Bus - MODBUS TCP *)

	EO_GENERIC		:=9000, (* Generic dataset *)
	EO_EXPO			:=9001  (* EXPO dataset *)
);
END_TYPE

(* Data type *)
TYPE en_SYS_Status :
(
	S_UNKNOWN  := 0,
	S_STARTUP,
	S_INIT_RTC,
	S_INIT_VAR,
	S_AUTOTEST,
	S_RUNNING,
	S_SHUTDOWN,
	S_HALT
);
END_TYPE

(* Data type in LON/Enumerations *)
TYPE file_request_t :
(
	FR_NUL := -1,
	FR_OPEN_TO_SEND := 0,
	FR_OPEN_TO_RECEIVE := 1,
	FR_CLOSE_FILE := 2,
	FR_CLOSE_DELETE_FILE := 3,
	FR_DIRECTORY_LOOKUP := 4,
	FR_OPEN_TO_SEND_RA := 5,
	FR_OPEN_TO_RECEIVE_RA := 6
);
END_TYPE

(* Data type in LON/Enumerations *)
TYPE file_status_t :
(
	FS_NUL := -1,
	FS_XFER_OK := 0,
	FS_LOOKUP_OK := 1,
	FS_OPEN_FAIL := 2,
	FS_LOOKUP_ERR := 3,
	FS_XFER_UNDERWAY := 4,
	FS_IO_ERR := 5,
	FS_TIMEOUT_ERR := 6,
	FS_WINDOW_ERR := 7,
	FS_AUTH_ERR := 8,
	FS_ACCESS_UNAVAIL := 9,
	FS_SEEK_INVALID := 10,
	FS_SEEK_WAIT := 11
);
END_TYPE

(* Data type in LON/Enumerations *)
TYPE hvac_t :
(
	HVAC_NUL := -1,
	HVAC_AUTO := 0,
	HVAC_HEAT := 1,
	HVAC_MRNG_WRMUP := 2,
	HVAC_COOL := 3,
	HVAC_NIGHT_PURGE := 4,
	HVAC_PRE_COOL := 5,
	HVAC_OFF := 6,
	HVAC_TEST := 7,
	HVAC_EMERG_HEAT := 8,
	HVAC_FAN_ONLY := 9,
	HVAC_FREE_COOL := 10,
	HVAC_ICE := 11,
	HVAC_MAX_HEAT := 12,
	HVAC_ECONOMY := 13,
	HVAC_DEHUMID := 14,
	HVAC_CALIBRATE := 15,
	HVAC_EMERG_COOL := 16,
	HVAC_EMERG_STEAM := 17,
	HVAC_MAX_COOL := 18,
	HVAC_HVC_LOAD := 19,
	HVAC_NO_LOAD := 20
);
END_TYPE

(* Data type in LON/Enumerations *)
TYPE object_request_t :
(
	RQ_NUL := -1,
	RQ_NORMAL := 0,
	RQ_DISABLED := 1,
	RQ_UPDATE_STATUS := 2,
	RQ_SELF_TEST := 3,
	RQ_UPDATE_ALARM := 4,
	RQ_REPORT_MASK := 5,
	RQ_OVERRIDE := 6,
	RQ_ENABLE := 7,
	RQ_RMV_OVERRIDE := 8,
	RQ_CLEAR_STATUS := 9,
	RQ_CLEAR_ALARM := 10,
	RQ_ALARM_NOTIFY_ENABLED := 11,
	RQ_ALARM_NOTIFY_DISABLED := 12,
	RQ_MANUAL_CTRL := 13,
	RQ_REMOTE_CTRL := 14,
	RQ_PROGRAM := 15,
	RQ_CLEAR_RESET := 16,
	RQ_RESET := 17,
	RQ_CLEAR_LOG := 18,
	RQ_LOAD_PROGRAM := 19,
	RQ_RUN_PROGRAM := 20,
	RQ_HALT_PROGRAM := 21,
	RQ_RESTART_PROGRAM := 22,
	RQ_UNLOAD_PROGRAM := 23,
	RQ_STEP_PROGRAM := 24
);
END_TYPE

(* Data type in LON/Enumerations *)
TYPE priority_level_t :
(
	PR_NUL := -1,
	PR_LEVEL_0 := 0,
	PR_LEVEL_1 := 1,
	PR_LEVEL_2 := 2,
	PR_LEVEL_3 := 3,
	PR_1 := 4,
	PR_2 := 5,
	PR_3 := 6,
	PR_4 := 7,
	PR_6 := 8,
	PR_8 := 9,
	PR_10 := 10,
	PR_16 := 11
);
END_TYPE

(* Data type in Plant_Objects *)
TYPE typ_Clima : (* CURVA CLIMATICA *)
STRUCT
	InitOK:		BOOL;
	Points: 	ARRAY [0..10] OF POINT;
END_STRUCT
END_TYPE

(* Data type in Plant_Objects *)
TYPE typ_Cron_Calendar :
STRUCT
	Profile		: ARRAY[0..384] OF BYTE;
END_STRUCT
END_TYPE

(* Data type in Plant_Objects *)
TYPE typ_Cron_Jolly :
STRUCT
	Start		: DT;
	End			: DT;
	Temp		: WORD;
	Flags		: WORD; (* B0:Enabled B1..B15:Unused *)
END_STRUCT
END_TYPE

(* Data type in Plant_Objects *)
TYPE typ_Cron_Profile :
STRUCT
	Flags		: WORD;
	Setpoint	: ARRAY [0..95] OF WORD;
END_STRUCT
END_TYPE

(* Data type in Errors *)
TYPE typ_Logger :
STRUCT
	Status		: en_Logger_Status;

	SendReq		: BOOL;
	SendIdx		: DWORD;
	SendData	: ARRAY [0..MAX_SEND_TCP_CLIENT] OF BYTE;
	SendLen		: DINT;

	TData		: ARRAY [0..MAX_SEND_TCP_CLIENT] OF BYTE;
	TLen		: DINT;

	LastIdxPos	: DWORD;

	(* Temporary variables used by objects *)
	s1			: STRING(256);
	i1			: WORD;

END_STRUCT
END_TYPE

(* Data type in Plant_Objects *)
TYPE typ_MODBUS_VAR : (* Gestione parametri MODBUS *)
STRUCT
	SlaveAddress	: BYTE;
	FunCode			: BYTE;
	FunAddress		: WORD;
	Refresh_Time	: BYTE; (* 0:No refresh x:Refresh in seconds *)
	Refresh_Cnt		: BYTE; (* INTERNAL *)
	Variable		: POINTER TO WORD;
	Variable_Size	: BYTE;
	Variable_Mirror : WORD; (* INTERNAL [Force refresh on read variables when <>0] *)
END_STRUCT
END_TYPE

(* Data type *)
TYPE typ_SYS :
STRUCT
	Status			: en_SYS_Status;
	Warning			: BOOL;
	Alarm			: BOOL;
	AlarmStop		: BOOL;

	Time_LogString	: STRING;
	Time_Year		: WORD;
	Time_Month		: BYTE;
	Time_Day		: BYTE;

	Time_CT_DT		: DT;
	Time_CT_Day		: WORD;
	Time_CT_Quarter	: BYTE;

	LastLogs_Idx	: BYTE;
	LastLogs_Dat	: ARRAY[0..5] OF STRING;
	LastLogs_Msg	: ARRAY[0..5] OF STRING;

END_STRUCT
END_TYPE

(* Data type in LON/NetworkVariables *)
TYPE typSnvtAlarm : 
STRUCT
	abLocation : ARRAY[0..5] OF BYTE;
	wObjectId : WORD;
	bAlarmType : BYTE (* enum type alarm_type_t *);
	bPriorityLevel : BYTE (* enum type priority_level_t *);
	wIndexToSnvt : WORD;
	abValue : ARRAY[0..3] OF BYTE;
	wYear : WORD;
	bMonth : BYTE;
	bDay : BYTE;
	bHour : BYTE;
	bMinute : BYTE;
	bSecond : BYTE;
	wMillisecond : WORD;
	abAlarmLimit : ARRAY[0..3] OF BYTE;
	bStatusInformation : BYTE; (* bit allocation of bStatusInformation:
	bit 0: NVI update counter LSB
	bit 1: NVI update counter
	bit 2: NVI update counter
	bit 3: NVI update counter MSB
	bit 4: timeout for NVI occurs (MaxRcvTime expired)
	bit 5: reserved
	bit 6: reserved
	bit 7: force NVO update *)
	bInternalUseOnly : BYTE; (* Do not use this byte in your application! *)
END_STRUCT
END_TYPE

(* Data type in LON/NetworkVariables *)
TYPE typSnvtFilePos : 
STRUCT
	diRwPtr : DINT;
	wRwLength : WORD;
	bStatusInformation : BYTE; (* bit allocation of bStatusInformation:
	bit 0: NVI update counter LSB
	bit 1: NVI update counter
	bit 2: NVI update counter
	bit 3: NVI update counter MSB
	bit 4: timeout for NVI occurs (MaxRcvTime expired)
	bit 5: reserved
	bit 6: reserved
	bit 7: force NVO update *)
	bInternalUseOnly : BYTE; (* Do not use this byte in your application! *)
END_STRUCT
END_TYPE

(* Data type in LON/NetworkVariables *)
TYPE typSnvtFileReq : 
STRUCT
	bRequest : BYTE (* enum type file_request_t *);
	wIndex : WORD;
	wReceiveTimeout : WORD;
	abDestAddress : ARRAY[0..4] OF BYTE (* union declaration *);
	bAuthOn : BYTE;
	bPrioOn : BYTE;
	bStatusInformation : BYTE; (* bit allocation of bStatusInformation:
	bit 0: NVI update counter LSB
	bit 1: NVI update counter
	bit 2: NVI update counter
	bit 3: NVI update counter MSB
	bit 4: timeout for NVI occurs (MaxRcvTime expired)
	bit 5: reserved
	bit 6: reserved
	bit 7: force NVO update *)
	bInternalUseOnly : BYTE; (* Do not use this byte in your application! *)
END_STRUCT
END_TYPE

(* Data type in LON/NetworkVariables *)
TYPE typSnvtFileStatus : 
STRUCT
	bStatus : BYTE (* enum type file_status_t *);
	wNumberOfFiles : WORD;
	wSelectedFile : WORD;
	abAdr : ARRAY[0..21] OF BYTE (* union declaration *);
	bStatusInformation : BYTE; (* bit allocation of bStatusInformation:
	bit 0: NVI update counter LSB
	bit 1: NVI update counter
	bit 2: NVI update counter
	bit 3: NVI update counter MSB
	bit 4: timeout for NVI occurs (MaxRcvTime expired)
	bit 5: reserved
	bit 6: reserved
	bit 7: force NVO update *)
	bInternalUseOnly : BYTE; (* Do not use this byte in your application! *)
END_STRUCT
END_TYPE

(* Data type in LON/NetworkVariables *)
TYPE typSnvtHvacMode : 
STRUCT
	bSnvtHvacMode : BYTE (* enum type hvac_t *);
	bStatusInformation : BYTE; (* bit allocation of bStatusInformation:
	bit 0: NVI update counter LSB
	bit 1: NVI update counter
	bit 2: NVI update counter
	bit 3: NVI update counter MSB
	bit 4: timeout for NVI occurs (MaxRcvTime expired)
	bit 5: reserved
	bit 6: reserved
	bit 7: force NVO update *)
	bInternalUseOnly : BYTE; (* Do not use this byte in your application! *)
END_STRUCT
END_TYPE

(* Data type in LON/NetworkVariables *)
TYPE typSnvtObjRequest : 
STRUCT
	wObjectId : WORD;
	bObjectRequest : BYTE (* enum type object_request_t *);
	bStatusInformation : BYTE; (* bit allocation of bStatusInformation:
	bit 0: NVI update counter LSB
	bit 1: NVI update counter
	bit 2: NVI update counter
	bit 3: NVI update counter MSB
	bit 4: timeout for NVI occurs (MaxRcvTime expired)
	bit 5: reserved
	bit 6: reserved
	bit 7: force NVO update *)
	bInternalUseOnly : BYTE; (* Do not use this byte in your application! *)
END_STRUCT
END_TYPE

(* Data type in LON/NetworkVariables *)
TYPE typSnvtObjStatus : 
STRUCT
	wObjectId : WORD;
	bBitfieldByteOffset2 : BYTE (* bit field *);
	bBitfieldByteOffset3 : BYTE (* bit field *);
	bBitfieldByteOffset4 : BYTE (* bit field *);
	bBitfieldByteOffset5 : BYTE (* bit field *);
	bStatusInformation : BYTE; (* bit allocation of bStatusInformation:
	bit 0: NVI update counter LSB
	bit 1: NVI update counter
	bit 2: NVI update counter
	bit 3: NVI update counter MSB
	bit 4: timeout for NVI occurs (MaxRcvTime expired)
	bit 5: reserved
	bit 6: reserved
	bit 7: force NVO update *)
	bInternalUseOnly : BYTE; (* Do not use this byte in your application! *)
END_STRUCT
END_TYPE

(* Data type in LON/NetworkVariables *)
TYPE typSnvtState : 
STRUCT
	bBitfieldByteOffset0 : BYTE (* bit field *);
	bBitfieldByteOffset1 : BYTE (* bit field *);
	bStatusInformation : BYTE; (* bit allocation of bStatusInformation:
	bit 0: NVI update counter LSB
	bit 1: NVI update counter
	bit 2: NVI update counter
	bit 3: NVI update counter MSB
	bit 4: timeout for NVI occurs (MaxRcvTime expired)
	bit 5: reserved
	bit 6: reserved
	bit 7: force NVO update *)
	bInternalUseOnly : BYTE; (* Do not use this byte in your application! *)
END_STRUCT
END_TYPE

(* Data type in LON/NetworkVariables *)
TYPE typSnvtSwitch : 
STRUCT
	bValue : BYTE;
	siState : SINT;
	bStatusInformation : BYTE; (* bit allocation of bStatusInformation:
	bit 0: NVI update counter LSB
	bit 1: NVI update counter
	bit 2: NVI update counter
	bit 3: NVI update counter MSB
	bit 4: timeout for NVI occurs (MaxRcvTime expired)
	bit 5: reserved
	bit 6: reserved
	bit 7: force NVO update *)
	bInternalUseOnly : BYTE; (* Do not use this byte in your application! *)
END_STRUCT
END_TYPE

(* Data type in LON/NetworkVariables *)
TYPE typSnvtTempP :
STRUCT
	iSnvtTempP : INT;
	bStatusInformation : BYTE; (* bit allocation of bStatusInformation:
	bit 0: NVI update counter LSB
	bit 1: NVI update counter
	bit 2: NVI update counter
	bit 3: NVI update counter MSB
	bit 4: timeout for NVI occurs (MaxRcvTime expired)
	bit 5: reserved
	bit 6: reserved
	bit 7: force NVO update *)
	bInternalUseOnly : BYTE; (* Do not use this byte in your application! *)
END_STRUCT
END_TYPE

(* Data type in LON/NetworkVariables *)
TYPE typSnvtTimeStamp : 
STRUCT
	iYear : INT;
	bMonth : BYTE;
	bDay : BYTE;
	bHour : BYTE;
	bMinute : BYTE;
	bSecond : BYTE;
	bStatusInformation : BYTE; (* bit allocation of bStatusInformation:
	bit 0: NVI update counter LSB
	bit 1: NVI update counter
	bit 2: NVI update counter
	bit 3: NVI update counter MSB
	bit 4: timeout for NVI occurs (MaxRcvTime expired)
	bit 5: reserved
	bit 6: reserved
	bit 7: force NVO update *)
	bInternalUseOnly : BYTE; (* Do not use this byte in your application! *)
END_STRUCT
END_TYPE

(* POU PLC_PRG, ST *)
PROGRAM PLC_PRG
VAR
	Timer1: TON; (* Fast controls tick *)
	Timer2: TON; (* Plant control tick *)
	Timer3: TON; (* Logger timer *)
END_VAR
(******************************************************************************
 ****                           MAIN TASK CODE                             ****
 ******************************************************************************

	Network setup:
		IP  = 192.168.100.2 | MSK = 255.255.255.0
		GW	= 192.168.100.1 | DNS = 192.168.100.1
		SNTP = 193.204.114.232 (3600s) ==> 192.168.100.3
*)

(*==============================*)
(*===== Main status machine ====*)
(*==============================*)
Main_Stm();

(*==============================*)
(*== Running cycle operations ==*)
(*==============================*)
IF SYS.Status>S_INIT_VAR THEN

	(* Update LON output variables (needs to be here to obtain only one refresh) *)
	CAL01.Heartbeat( CLIM:=CAL01_Clima );
	(* Execute LON process *)
	Module_1_PRG();

END_IF

(*==============================*)
(*== System cycle operations ===*)
(*==============================*)
(* Execute TCP processes *)
Logger_Proc();
Remote_Proc();
(* Update user led *)
USRLED_Update();
(* Execute Cron Editor commands *)
CronEd();
(* External resources *)
IF TPV01.ERR THEN T_AMB:=Plant_DefaultTAmb; ELSE T_AMB:=T_S01; END_IF
END_PROGRAM
ACTION Main_Stm:
CASE Sys.Status OF

	S_STARTUP:
		Sys.Status:=S_INIT_RTC;

	S_INIT_RTC:
		(* Check RTC and update from network *)
		RTC_Update();
		(* Check time *)
		IF Sys.Time_Year>2000 THEN
			Sys.Status:=S_INIT_VAR;
		END_IF

	S_INIT_VAR:
		LogEv(EL_Wrn,EO_SYS,0,1,CONCAT('System_startup_v',WORD_TO_STRING(Plant_SW_VER)));
		Sys.Status:=S_RUNNING;

	S_RUNNING:
		Timer1(IN:=NOT Timer1.Q,PT:=T#50ms);
		IF Timer1.Q THEN
			(* Update meters *)
			CTL01 ( CTL_ST:=CTL01_ST, COUNT:=CTL01_Count );
			(* Update system checks *)
			SYS_Proc();
		END_IF

		Timer2(IN:=NOT Timer2.Q,PT:=T#500ms);
		IF Timer2.Q THEN
			(* Read current date/time *)
			RTC_Update();
			(* Execute plant operations *)
			TPV01	 ( IN:=T_S01 );
			TPV02	 ( IN:=(CAL01.CFD_Temp.iSnvtTempP/10) );
			TPV03	 ( IN:=T_S03 );
			TPV04	 ( IN:=T_S04 );
			TPV05	 ( IN:=T_S05 );
			CRON01( SETPOINT=>CIR01.Ctrl_SetPoint );
			CRON02( SETPOINT=>CIR02.Ctrl_SetPoint );
			CRON03( SETPOINT=>CIR03.Ctrl_SetPoint );
			CRON04( SETPOINT=>CIR04.Ctrl_SetPoint );
			CRON05( SETPOINT=>CIR05.Ctrl_SetPoint );
			CRON06( SETPOINT=>CIR06.Ctrl_SetPoint );
			CRON07( SETPOINT=>CIR07.Ctrl_SetPoint );
			CRON08( SETPOINT=>CIR08.Ctrl_SetPoint );
			CRON09( SETPOINT=>CIR09.Ctrl_SetPoint );
			CIR01 ( CIR_AL:=CIR01_AL     , CIR_ST:=CIR01_ST , CIR_STOP_REQ:=FALSE        , CIR_EN=>CIR01_EN );
			CIR02 ( CIR_AL:=NOT CIR02_AL , CIR_ST:=CIR02_ST , CIR_STOP_REQ:=VRD01.Alarm1 , CIR_EN=>CIR02_EN );
			CIR03 ( CIR_AL:=NOT CIR03_AL , CIR_ST:=CIR03_ST , CIR_STOP_REQ:=FALSE        , CIR_EN=>CIR03_EN );
			CIR04 ( CIR_AL:=NOT CIR04_AL , CIR_ST:=CIR04_ST , CIR_STOP_REQ:=FALSE        , CIR_EN=>CIR04_EN );
			CIR05 ( CIR_AL:=NOT CIR05_AL , CIR_ST:=CIR05_ST , CIR_STOP_REQ:=FALSE        , CIR_EN=>CIR05_EN );
			CIR06 ( CIR_AL:=NOT CIR06_AL , CIR_ST:=CIR06_ST , CIR_STOP_REQ:=VRD02.Alarm1 , CIR_EN=>CIR06_EN );
			CIR07 ( CIR_AL:=NOT CIR07_AL , CIR_ST:=CIR07_ST , CIR_STOP_REQ:=FALSE        , CIR_EN=>CIR07_EN );
			CIR08 ( CIR_AL:=NOT CIR08_AL , CIR_ST:=CIR08_ST , CIR_STOP_REQ:=FALSE        , CIR_EN=>CIR08_EN );
			CIR09 ( CIR_AL:=NOT CIR09_AL , CIR_ST:=CIR09_ST , CIR_STOP_REQ:=FALSE        , CIR_EN=>CIR09_EN );
			VRD01 ( CLIM:=VRD01_Clima , TEMP:=T_S04 , STATUS:=VRD01_ST , RUN:=CIR02_EN ,	OUT=>VRD01_CTRL );
			VRD02 ( CLIM:=VRD02_Clima , TEMP:=T_S05 , STATUS:=VRD02_ST , RUN:=CIR06_EN ,	OUT=>VRD02_CTRL );
			CAL01.Run:=( CIR01.Run OR CIR02.Run OR CIR03.Run OR CIR04.Run OR CIR05.Run OR
						 CIR06.Run OR CIR07.Run OR CIR08.Run OR CIR09.Run ) AND SYS.AlarmStop=FALSE;
			CAL01 ( CLIM:=CAL01_Clima );
			(* Test toggle *)
			IF TEST1 THEN TEST1:=FALSE; ELSE TEST1:=TRUE; END_IF
		END_IF

		Timer3(IN:=NOT Timer3.Q,PT:=T#5m);
		IF Timer3.Q THEN
			(* Trig logger *)
			LogTrig();
			(* Execute temporary CSV logger *)
			CSV_Log();
		END_IF

	S_SHUTDOWN:
		(* Stop caldaia *)
		(* Stop deviatori *)
		(* Aspetta 5 min prima di spegnere eventuali circolatori *)
		Sys.Status:=S_STARTUP;

	S_HALT:
		(* Aspetta uscita manuale *)
		Sys.Status:=S_STARTUP;


ELSE
	Sys.Status:=S_STARTUP;
END_CASE;
END_ACTION

(* POU LON/Module_1/Module_1_PRG, FBD *)
PROGRAM Module_1_PRG
VAR
	(* Automatic added code, do not change! *)
	LonMaster : Module_1_LonMaster;
	SFPTnodeObject : Module_1_SFPTnodeObject;
	Virtualfunctionalblock : Module_1_Virtualfunctionalblock;

	InData_LON AT %IB8 : ARRAY[0..23] OF BYTE;
	OutData_LON AT %QB0 : ARRAY[0..23] OF BYTE;
	(***** End of automatic added code. *****)

	(* Add your code here. *)

	LonState: BOOL;
	LonReset: BOOL;
END_VAR
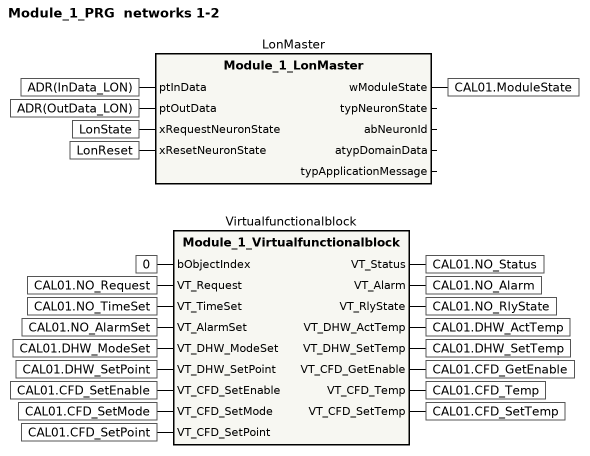
_FBD_ (* Function Block Diagram *)
NETWORK 1 (* Added by code generator *)
	LonMaster:Module_1_LonMaster(ptInData: ADR(InData_LON), ptOutData: ADR(OutData_LON), xRequestNeuronState: LonState, xResetNeuronState: LonReset) => CAL01.ModuleState
NETWORK 2
	Virtualfunctionalblock:Module_1_Virtualfunctionalblock(bObjectIndex: 0, VT_Request: CAL01.NO_Request, VT_TimeSet: CAL01.NO_TimeSet, VT_AlarmSet: CAL01.NO_AlarmSet, VT_DHW_ModeSet: CAL01.DHW_ModeSet, VT_DHW_SetPoint: CAL01.DHW_SetPoint, VT_CFD_SetEnable: CAL01.CFD_SetEnable, VT_CFD_SetMode: CAL01.CFD_SetMode, VT_CFD_SetPoint: CAL01.CFD_SetPoint, VT_Alarm => CAL01.NO_Alarm, VT_RlyState => CAL01.NO_RlyState, VT_DHW_ActTemp => CAL01.DHW_ActTemp, VT_DHW_SetTemp => CAL01.DHW_SetTemp, VT_CFD_GetEnable => CAL01.CFD_GetEnable, VT_CFD_Temp => CAL01.CFD_Temp, VT_CFD_SetTemp => CAL01.CFD_SetTemp) => CAL01.NO_Status
_END_FBD_
(* the same logic as Structured Text *)
(* Network 1: Added by code generator *)
LonMaster(ptInData := ADR(InData_LON), ptOutData := ADR(OutData_LON), xRequestNeuronState := LonState, xResetNeuronState := LonReset);
CAL01.ModuleState := LonMaster.wModuleState;
(* Network 2 *)
Virtualfunctionalblock(bObjectIndex := 0, VT_Request := CAL01.NO_Request, VT_TimeSet := CAL01.NO_TimeSet, VT_AlarmSet := CAL01.NO_AlarmSet, VT_DHW_ModeSet := CAL01.DHW_ModeSet, VT_DHW_SetPoint := CAL01.DHW_SetPoint, VT_CFD_SetEnable := CAL01.CFD_SetEnable, VT_CFD_SetMode := CAL01.CFD_SetMode, VT_CFD_SetPoint := CAL01.CFD_SetPoint);
CAL01.NO_Alarm := Virtualfunctionalblock.VT_Alarm;
CAL01.NO_RlyState := Virtualfunctionalblock.VT_RlyState;
CAL01.DHW_ActTemp := Virtualfunctionalblock.VT_DHW_ActTemp;
CAL01.DHW_SetTemp := Virtualfunctionalblock.VT_DHW_SetTemp;
CAL01.CFD_GetEnable := Virtualfunctionalblock.VT_CFD_GetEnable;
CAL01.CFD_Temp := Virtualfunctionalblock.VT_CFD_Temp;
CAL01.CFD_SetTemp := Virtualfunctionalblock.VT_CFD_SetTemp;
CAL01.NO_Status := Virtualfunctionalblock.VT_Status;
END_PROGRAM

(* POU LON/Module_1/Master/Module_1_LonMaster, ST *)
FUNCTION_BLOCK Module_1_LonMaster
(******************************************)
(* Automatic generated code, do not edit! *)
(******************************************)
VAR_INPUT
	ptInData  : POINTER TO BYTE;
	ptOutData : POINTER TO BYTE;
	xRequestNeuronState : BOOL;
	xResetNeuronState : BOOL;
END_VAR
VAR_OUTPUT
	wModuleState : WORD; (* bit coded wModuleState:
	15: communication to I/O-module interrupted (error)
	14 - 08: reserved
	07: ready for Neuron initialization
	06: Neuron active
	05: user interface active
	04: internal module communication interrupted (error)
	03: CP synchronization running
	02: Neuron is configured online
	01 - 00: reserved *)

	typNeuronState : NeuronState;
	abNeuronId : ARRAY[0..5] OF BYTE;
	atypDomainData : ARRAY[0..1] OF DomainData;
	typApplicationMessage : ApplicationMessageData;
END_VAR
VAR
	bInternalCode : BYTE;
	bNvIndex : BYTE;
	wCpIndex : WORD;
	lonCom : FbLonBasicCommunication;

	xInitIsStarted : BOOL := FALSE;

	TimeoutTimer : TON;
	timeOutTime : TIME := T#1000ms;
	xStateMachineIsChecked : BOOL;
	xTimerStart : BOOL;

	iDomainTable : INT;
	xSendRequestPending : BOOL;
	trigRequest : R_TRIG;
	trigReset : R_TRIG;

	abMbxRxPrio0Buf: ARRAY [0..309] OF BYTE;
	abMbxRxPrio1Buf: ARRAY [0..517] OF BYTE;
	aMbxRxBufSize: ARRAY [0..1] OF UINT := 310, 518;
	aMbxRxBufList: ARRAY [0..1] OF POINTER TO BYTE;
	afbMbxRxFb: ARRAY [0..1] OF MBX2_RX_DEFRAG;
	astMbxRxCtx: ARRAY [0..1] OF stMbx2DefragContext;

	abMbxTxPrio0Buf: ARRAY [0..309] OF BYTE;
	abMbxTxPrio1Buf: ARRAY [0..517] OF BYTE;
	aMbxTxBufSize: ARRAY [0..1] OF UINT := 310, 518;
	aMbxTxBufList: ARRAY [0..1] OF POINTER TO BYTE;
	afbMbxTxFb: ARRAY [0..1] OF MBX2_TX_FRAG;

	astMbxTrackContext: ARRAY [0..0] OF stMbx2TrackContext;
END_VAR
VAR CONSTANT
END_VAR
aMbxRxBufList[0] := ADR(abMbxRxPrio0Buf[0]);
aMbxRxBufList[1] := ADR(abMbxRxPrio1Buf[0]);

aMbxTxBufList[0] := ADR(abMbxTxPrio0Buf[0]);
aMbxTxBufList[1] := ADR(abMbxTxPrio1Buf[0]);

mbxModule_1.Ressources.pDefragBufList := ADR(aMbxRxBufList);
mbxModule_1.Ressources.pDefragBufSizeList := ADR(aMbxRxBufSize);
mbxModule_1.Ressources.pDefragCtxPtrList := ADR(astMbxRxCtx);
mbxModule_1.Ressources.pDefragFbList := ADR(afbMbxRxFb);
mbxModule_1.Ressources.pFragBufList := ADR(aMbxTxBufList);
mbxModule_1.Ressources.pFragBufSizeList := ADR(aMbxTxBufSize);
mbxModule_1.Ressources.pFragFbList := ADR(afbMbxTxFb);

mbxModule_1.Ressources.unMaxAvailableRxPrioIndex := 1;
mbxModule_1.Ressources.unMaxAvailableTxPrioIndex := 1;

mbxModule_1.Ressources.pTrackStList := ADR(astMbxTrackContext);
mbxModule_1.Ressources.unMaxAvailableTrackIndex := 0;

mbxModule_1.Ressources.pabRxWin := ptInData + 1;
mbxModule_1.Ressources.pabTxWin := ptOutData + 1;
mbxModule_1.Ressources.bTxWinSize := 23;
mbxModule_1.Ressources.bRxWinSize := 23;

IF (mbxModule_1.bStatus.2 = TRUE) OR (mbxModule_1.bStatus.1 = TRUE) THEN
	mbxModule_1.MBX_RESET();
	xInitRunning_Module_1 := TRUE;
	xInitIsStarted := FALSE;
END_IF
mbxModule_1.MBX_CYCLE();

IF (mbxModule_1.bStatus.0 <> TRUE) THEN 
	wModuleState := 16#8000;
	RETURN;
ELSE
	wModuleState.15 := FALSE;
END_IF

xStateMachineIsChecked := FALSE;
IF xInitRunning_Module_1 = TRUE THEN
	IF xInitIsStarted = FALSE THEN
		SetParameter();
		lonCom.eInitState := INIT_SND_SGNTR_REQ;
		lonCom.CheckInitState();
		xInitIsStarted := TRUE;
		xStateMachineIsChecked := TRUE;
	END_IF
END_IF

typApplicationMessage.xMsgRcvd := FALSE;
typApplicationMessage.xRspRcvd := FALSE;
ResetNviUpdate();
WHILE (mbxModule_1.xRxPending) DO
	unLastLen_mbxModule_1 := mbxModule_1.unRxLen;
	mbxModule_1.pbRxData := ADR(InDataTelegram_Module_1);
	mbxModule_1.MBX_RETRIEVE();
	IF (mbxModule_1.nError <> MBX_OK) THEN EXIT; END_IF;
	bInternalCode := InDataTelegram_Module_1[0];

	IF (xInitRunning_Module_1 = TRUE) AND (lonCom.eInitState <> INIT_TRANSFER_CFG) THEN
		IF (FuCheckForValidInitCode(bInternalCode)) THEN
			SetParameter();
			lonCom.unLastLen := unLastLen_mbxModule_1;
			lonCom.CheckInitState();
			xInitRunning_Module_1 := NOT lonCom.xInitDone;
			xStateMachineIsChecked := TRUE;
		END_IF
	END_IF

	IF (bInternalCode = M2C_NVI_UPDT_OCCD) OR (bInternalCode = M2C_NV_VALUE_RSP) OR (bInternalCode = M2C_NVI_UPDT_TOUT) THEN
		bNvIndex := InDataTelegram_Module_1[1];
		CASE bNvIndex OF
			0, 2, 4: Module_1_PRG.SFPTnodeObject.DataReceived();
			6, 8, 10, 12, 14, 16, 18, 20: Module_1_PRG.Virtualfunctionalblock.DataReceived();

		END_CASE;
	ELSIF (bInternalCode = M2C_CP_VALUE_RSP) THEN
		wCpIndex := InDataTelegram_Module_1[1] OR (InDataTelegram_Module_1[2] * 256);
		CASE wCpIndex OF

		END_CASE;
	ELSIF (bInternalCode = M2C_LON_MSG_RCVD) OR (bInternalCode = M2C_LON_RSP_RCVD) THEN
		ApplMsgReceived();
	ELSIF (bInternalCode = M2C_STATUS_RSP) THEN
		wModuleState := (wModuleState AND 16#FF00) + InDataTelegram_Module_1[1];
	ELSIF (bInternalCode = M2C_NEURON_ID) THEN
		FuMemCopy(ADR(InDataTelegram_Module_1[1]), ADR(abNeuronId), 6);
	ELSIF (bInternalCode = M2C_DOMAIN_DATA) THEN
		DomainDataRcvd();
	ELSIF (bInternalCode = M2C_MICRO_SERVER_STATUS_RSP) THEN
		NeuronStateRcvd();
	END_IF
END_WHILE

IF (xInitRunning_Module_1 = TRUE) AND ((lonCom.xCallStateMachine = TRUE) OR (TimeoutTimer.Q = TRUE)) AND (NOT xStateMachineIsChecked) THEN
	SetParameter();
	lonCom.xTimeOut := TimeoutTimer.Q;
	lonCom.CheckInitState();
END_IF
TimeoutTimer(IN:=lonCom.xTimerStart, PT:=timeOutTime);

trigRequest(CLK := xRequestNeuronState);
trigReset(CLK := xResetNeuronState);
IF (trigRequest.Q OR trigReset.Q) THEN
	RequestNeuronState();
END_IF
END_FUNCTION_BLOCK
ACTION ApplMsgReceived:
IF (InDataTelegram_Module_1[0] = M2C_LON_MSG_RCVD) THEN
	typApplicationMessage.typService := InDataTelegram_Module_1[1] AND 16#30;
	typApplicationMessage.bSourceSubnetId := InDataTelegram_Module_1[2];
	typApplicationMessage.bSourceNodeId := InDataTelegram_Module_1[3];
	typApplicationMessage.bCorrelator := InDataTelegram_Module_1[4];
	typApplicationMessage.bCode :=  InDataTelegram_Module_1[5];
	typApplicationMessage.bDataLength := UINT_TO_BYTE(unLastLen_mbxModule_1 - 6);
	IF typApplicationMessage.bDataLength > 48 THEN typApplicationMessage.bDataLength := 48; END_IF;
	FuMemSet(ADR(typApplicationMessage.abData), 0, SIZEOF(typApplicationMessage.abData));
	IF typApplicationMessage.bDataLength > 0 THEN
		FuMemCopy(ADR(InDataTelegram_Module_1[6]), ADR(typApplicationMessage.abData), typApplicationMessage.bDataLength);
	END_IF
	typApplicationMessage.xMsgRcvd := TRUE;
ELSE
	typApplicationMessage.typService := LON_RESPONSE;
	typApplicationMessage.bSourceSubnetId := InDataTelegram_Module_1[1];
	typApplicationMessage.bSourceNodeId := InDataTelegram_Module_1[2];
	typApplicationMessage.bCorrelator := 0;
	typApplicationMessage.bCode :=  InDataTelegram_Module_1[3];
	typApplicationMessage.bDataLength := UINT_TO_BYTE(unLastLen_mbxModule_1 - 4);
	IF typApplicationMessage.bDataLength > 48 THEN typApplicationMessage.bDataLength := 48; END_IF;
	FuMemSet(ADR(typApplicationMessage.abData), 0, SIZEOF(typApplicationMessage.abData));
	IF typApplicationMessage.bDataLength > 0 THEN
		FuMemCopy(ADR(InDataTelegram_Module_1[4]), ADR(typApplicationMessage.abData), typApplicationMessage.bDataLength);
	END_IF
	typApplicationMessage.xRspRcvd := TRUE;
END_IF
END_ACTION
ACTION DomainDataRcvd:
IF (unLastLen_mbxModule_1 = 17) THEN
	iDomainTable := InDataTelegram_Module_1[1];
	IF (iDomainTable < 0) OR (iDomainTable > 1) THEN RETURN; END_IF
	FuMemCopy(ADR(InDataTelegram_Module_1[2]), ADR(atypDomainData[iDomainTable].abDomainId), 6);
	atypDomainData[iDomainTable].bSubnet := InDataTelegram_Module_1[8];
	atypDomainData[iDomainTable].xIsNonClone := InDataTelegram_Module_1[9].7;
	atypDomainData[iDomainTable].bNodeId := InDataTelegram_Module_1[9] AND 16#7F;
	atypDomainData[iDomainTable].xIsInvalid := InDataTelegram_Module_1[10].7;
	atypDomainData[iDomainTable].bDomainIdLength := InDataTelegram_Module_1[10] AND 16#7F;
	FuMemCopy(ADR(InDataTelegram_Module_1[11]), ADR(atypDomainData[iDomainTable].abAuthenticationKey), 6);
END_IF
END_ACTION
ACTION NeuronStateRcvd:
IF (unLastLen_mbxModule_1 = 16) THEN
	typNeuronState.wCrcError := InDataTelegram_Module_1[1] + InDataTelegram_Module_1[2] * 256;
	typNeuronState.wTransactionTimeouts := InDataTelegram_Module_1[3] + InDataTelegram_Module_1[4] * 256;
	typNeuronState.wReceiveTransactionBuffersFull := InDataTelegram_Module_1[5] + InDataTelegram_Module_1[6] * 256;
	typNeuronState.wLostMessages := InDataTelegram_Module_1[7] + InDataTelegram_Module_1[8] * 256;
	typNeuronState.wMissedMessages := InDataTelegram_Module_1[9] + InDataTelegram_Module_1[10] * 256;
	typNeuronState.bResetCause := InDataTelegram_Module_1[11];
	typNeuronState.bNodeState := InDataTelegram_Module_1[12];
	typNeuronState.bFirmwareVersion := InDataTelegram_Module_1[13];
	typNeuronState.bLastErrorLogged := InDataTelegram_Module_1[14];
	typNeuronState.bModelNumber := InDataTelegram_Module_1[15];
END_IF
END_ACTION
ACTION RequestNeuronState:
OutDataTelegram_Module_1[0] := C2M_MICRO_SERVER_STATUS_QRY;
OutDataTelegram_Module_1[1] := BOOL_TO_BYTE(trigReset.Q);

mbxModule_1.bTxPrio := 1;
mbxModule_1.bTxProtID := 0;
mbxModule_1.pbTxData := ADR(OutDataTelegram_Module_1);
mbxModule_1.unTxLen := 2;
mbxModule_1.MBX_SEND();

IF (mbxModule_1.nError <> MBX_OK) THEN
	RETURN;
END_IF
END_ACTION
ACTION ResetNviUpdate:
Module_1_PRG.SFPTnodeObject.ResetNviUpdate();
Module_1_PRG.Virtualfunctionalblock.ResetNviUpdate();
END_ACTION
ACTION SetParameter:
lonCom.pMbx 			:= ADR(mbxModule_1);
lonCom.pInData 			:= ADR(InDataTelegram_Module_1);
lonCom.pOutData 		:= ADR(OutDataTelegram_Module_1);
lonCom.pTimer			:= ADR(TimeoutTimer);

lonCom.pActualSignature	:= ADR(abSignature_Module_1);
lonCom.pConfigBlock := ADR(abInterface_Module_1);
lonCom.wConfigSize 		:= wConfigSize_Module_1;
END_ACTION

(* POU LON/Module_1/NV_Interface/Module_1_SFPTnodeObject, ST *)
FUNCTION_BLOCK Module_1_SFPTnodeObject
(******************************************)
(* Automatic generated code, do not edit! *)
(******************************************)
VAR_INPUT
	bObjectIndex : BYTE := 0;
	nvoStatus : typSnvtObjStatus;
	nvoFileStat : typSnvtFileStatus;

END_VAR
VAR_OUTPUT
	nviRequest : typSnvtObjRequest;
	nviFileReq : typSnvtFileReq;
	nviFilePos : typSnvtFilePos;

END_VAR
VAR
	xSetOnce : BOOL := TRUE;
	xDataInUpdated : BOOL := FALSE;
	nvoStatusLast: typSnvtObjStatus;
	nvoFileStatLast: typSnvtFileStatus;

	cmd : BYTE;
	z : INT;
	bNvRelativeIdx : BYTE;
	bNvAbsoluteIdx : BYTE;
	wCpRelativeIdx : WORD;
	wCpAbsoluteIdx : WORD;
END_VAR
VAR CONSTANT
	bNvStartIndex : BYTE := 0;
	wCpStartIndex : WORD := 65535;
	bLmoCount : BYTE := 1;
END_VAR
IF (xInitRunning_Module_1 = TRUE) AND (xSetOnce = TRUE) THEN
	xSetOnce := FALSE;
	CachePointers();
	SetUpdateFlags();
END_IF

CheckUpdateFlags();
IF (xInitRunning_Module_1 = FALSE) AND (xDataInUpdated = FALSE) THEN
	IF (mbxModule_1.bStatus.0) THEN
		SendValueRequest();
	END_IF
END_IF

IF (xInitRunning_Module_1 = FALSE) AND (mbxModule_1.bStatus.0) THEN
	xSetOnce := TRUE;
	xDataInUpdated := FALSE;
	IF ((NOT FuMemCompare(ADR(nvoStatusLast), ADR(nvoStatus), ADR(nvoStatus.bStatusInformation) - ADR(nvoStatus))) OR (nvoStatus.bStatusInformation.7 = TRUE) OR (nvoStatusLast.bInternalUseOnly.1 = TRUE)) THEN
		FuSnvtObjStatusToRaw(ADR(nvoStatus), ADR(OutDataTelegram_Module_1[2]));

		bNvAbsoluteIdx := bNvStartIndex + bObjectIndex + (1 * bLmoCount);

		IF (FuDoNvoUpdate_Module_1(ADR(nvoStatus), ADR(nvoStatusLast), ADR(nvoStatus.bInternalUseOnly), ADR(nvoStatusLast.bInternalUseOnly), ADR(nvoStatus.bStatusInformation), bNvAbsoluteIdx, 6, SIZEOF(nvoStatus)) = FALSE) THEN
			RETURN;
		END_IF
	END_IF
	IF ((NOT FuMemCompare(ADR(nvoFileStatLast), ADR(nvoFileStat), ADR(nvoFileStat.bStatusInformation) - ADR(nvoFileStat))) OR (nvoFileStat.bStatusInformation.7 = TRUE) OR (nvoFileStatLast.bInternalUseOnly.1 = TRUE)) THEN
		FuSnvtFileStatusToRaw(ADR(nvoFileStat), ADR(OutDataTelegram_Module_1[2]));

		bNvAbsoluteIdx := bNvStartIndex + bObjectIndex + (3 * bLmoCount);

		IF (FuDoNvoUpdate_Module_1(ADR(nvoFileStat), ADR(nvoFileStatLast), ADR(nvoFileStat.bInternalUseOnly), ADR(nvoFileStatLast.bInternalUseOnly), ADR(nvoFileStat.bStatusInformation), bNvAbsoluteIdx, 27, SIZEOF(nvoFileStat)) = FALSE) THEN
			RETURN;
		END_IF
	END_IF

END_IF
END_FUNCTION_BLOCK
ACTION CachePointers:
;
END_ACTION
ACTION CheckUpdateFlags:
xDataInUpdated := (NOT nviRequest.bInternalUseOnly.0) AND (NOT nviFileReq.bInternalUseOnly.0) AND (NOT nviFilePos.bInternalUseOnly.0) AND TRUE;
END_ACTION
ACTION DataReceived:
cmd := InDataTelegram_Module_1[0];
IF (cmd = M2C_NVI_UPDT_OCCD) OR (cmd = M2C_NV_VALUE_RSP) OR (cmd = M2C_NVI_UPDT_TOUT) THEN
	bNvRelativeIdx := (InDataTelegram_Module_1[1] - bNvStartIndex - bObjectIndex) / bLmoCount;
	CASE bNvRelativeIdx OF
	0:
		IF (cmd = M2C_NVI_UPDT_OCCD) OR (cmd = M2C_NV_VALUE_RSP) THEN
			IF (unLastLen_mbxModule_1 = (2 + 3)) THEN
				FuRawToSnvtObjRequest(ADR(InDataTelegram_Module_1[2]), ADR(nviRequest));
				nviRequest.bInternalUseOnly.0 := FALSE;
				nviRequest.bStatusInformation := FuInkrementNviStatus(nviRequest.bStatusInformation);
			ELSIF (unLastLen_mbxModule_1 = 2) THEN
				nviRequest.bStatusInformation := FuInkrementNviStatus(nviRequest.bStatusInformation);
			END_IF
		ELSIF (cmd = M2C_NVI_UPDT_TOUT) THEN
			IF (unLastLen_mbxModule_1 = 3) THEN
				nviRequest.bStatusInformation.4 := BYTE_TO_BOOL(InDataTelegram_Module_1[2]);
			END_IF
		END_IF
	2:
		IF (cmd = M2C_NVI_UPDT_OCCD) OR (cmd = M2C_NV_VALUE_RSP) THEN
			IF (unLastLen_mbxModule_1 = (2 + 12)) THEN
				FuRawToSnvtFileReq(ADR(InDataTelegram_Module_1[2]), ADR(nviFileReq));
				nviFileReq.bInternalUseOnly.0 := FALSE;
				nviFileReq.bStatusInformation := FuInkrementNviStatus(nviFileReq.bStatusInformation);
			ELSIF (unLastLen_mbxModule_1 = 2) THEN
				nviFileReq.bStatusInformation := FuInkrementNviStatus(nviFileReq.bStatusInformation);
			END_IF
		ELSIF (cmd = M2C_NVI_UPDT_TOUT) THEN
			IF (unLastLen_mbxModule_1 = 3) THEN
				nviFileReq.bStatusInformation.4 := BYTE_TO_BOOL(InDataTelegram_Module_1[2]);
			END_IF
		END_IF
	4:
		IF (cmd = M2C_NVI_UPDT_OCCD) OR (cmd = M2C_NV_VALUE_RSP) THEN
			IF (unLastLen_mbxModule_1 = (2 + 6)) THEN
				FuRawToSnvtFilePos(ADR(InDataTelegram_Module_1[2]), ADR(nviFilePos));
				nviFilePos.bInternalUseOnly.0 := FALSE;
				nviFilePos.bStatusInformation := FuInkrementNviStatus(nviFilePos.bStatusInformation);
			ELSIF (unLastLen_mbxModule_1 = 2) THEN
				nviFilePos.bStatusInformation := FuInkrementNviStatus(nviFilePos.bStatusInformation);
			END_IF
		ELSIF (cmd = M2C_NVI_UPDT_TOUT) THEN
			IF (unLastLen_mbxModule_1 = 3) THEN
				nviFilePos.bStatusInformation.4 := BYTE_TO_BOOL(InDataTelegram_Module_1[2]);
			END_IF
		END_IF

	END_CASE
ELSIF (cmd = M2C_CP_VALUE_RSP) THEN
	wCpRelativeIdx := ((InDataTelegram_Module_1[1] + InDataTelegram_Module_1[2] * 256) - wCpStartIndex - bObjectIndex) / bLmoCount;
	CASE wCpRelativeIdx OF

	END_CASE
END_IF
END_ACTION
ACTION ResetNviUpdate:
nviRequest.bStatusInformation := nviRequest.bStatusInformation AND 16#F8;
nviFileReq.bStatusInformation := nviFileReq.bStatusInformation AND 16#F8;
nviFilePos.bStatusInformation := nviFilePos.bStatusInformation AND 16#F8;
;
END_ACTION
ACTION SendValueRequest:
IF (FuSendNviValueReq_Module_1(ADR(nviRequest.bInternalUseOnly), bNvStartIndex + bObjectIndex + (0 * bLmoCount)) = FALSE) THEN
	RETURN;
END_IF

IF (FuSendNviValueReq_Module_1(ADR(nviFileReq.bInternalUseOnly), bNvStartIndex + bObjectIndex + (2 * bLmoCount)) = FALSE) THEN
	RETURN;
END_IF

IF (FuSendNviValueReq_Module_1(ADR(nviFilePos.bInternalUseOnly), bNvStartIndex + bObjectIndex + (4 * bLmoCount)) = FALSE) THEN
	RETURN;
END_IF

;
END_ACTION
ACTION SetUpdateFlags:
nviRequest.bInternaluseOnly.0 := TRUE;
nvoStatusLast.bInternaluseOnly.1 := TRUE;
nvoStatusLast.bInternaluseOnly.7 := FALSE;
nviFileReq.bInternaluseOnly.0 := TRUE;
nvoFileStatLast.bInternaluseOnly.1 := TRUE;
nvoFileStatLast.bInternaluseOnly.7 := FALSE;
nviFilePos.bInternaluseOnly.0 := TRUE;
;
END_ACTION

(* POU LON/Shared/Internal/FuSnvtObjStatusToRaw, ST *)
FUNCTION FuSnvtObjStatusToRaw : BOOL
(******************************************)
(* Automatic generated code, do not edit! *)
(******************************************)
VAR_INPUT
	NvDataIn :  POINTER TO typSnvtObjStatus;
	DataOut : POINTER TO ARRAY[0..5] OF BYTE;
END_VAR
VAR
END_VAR
DataOut^[0] := WORD_TO_BYTE(SHR(NvDataIn^.wObjectId, 8));
DataOut^[1] := WORD_TO_BYTE(NvDataIn^.wObjectId);

DataOut^[2] := NvDataIn^.bBitfieldByteOffset2;

DataOut^[3] := NvDataIn^.bBitfieldByteOffset3;

DataOut^[4] := NvDataIn^.bBitfieldByteOffset4;

DataOut^[5] := NvDataIn^.bBitfieldByteOffset5;

FuSnvtObjStatusToRaw := TRUE;
END_FUNCTION

(* POU LON/Module_1/Internal/FuDoNvoUpdate_Module_1, ST *)
FUNCTION FuDoNvoUpdate_Module_1 : BOOL
(******************************************)
(* Automatic generated code, do not edit! *)
(******************************************)
VAR_INPUT
	ptNvo : POINTER TO BYTE;
	ptNvoLast : POINTER TO BYTE;
	ptNvoInternalUse : POINTER TO BYTE;
	ptNvoLastInternalUse : POINTER TO BYTE;
	ptNvoStatusInformation : POINTER TO BYTE;
	bNvoIndex : BYTE;
	uiNvoLength : UINT;
	uiNvoVariableLength : UINT;
END_VAR
IF (ptNvoLastInternalUse^.1 = TRUE) AND (ptNvoStatusInformation^.7 = FALSE) THEN
	OutDataTelegram_Module_1[0] := C2M_NV_VALUE;
ELSE
	OutDataTelegram_Module_1[0] := C2M_NVO_PROPAGATE;
END_IF
OutDataTelegram_Module_1[1] := bNvoIndex;

mbxModule_1.bTxPrio := BOOL_TO_BYTE(ptNvoLastInternalUse^.7);
mbxModule_1.bTxProtID := 0;
mbxModule_1.pbTxData := ADR(OutDataTelegram_Module_1);
mbxModule_1.unTxLen := 2 + uiNvoLength;
mbxModule_1.MBX_SEND();

IF (mbxModule_1.nError <> MBX_OK) THEN
	FuDoNvoUpdate_Module_1 := FALSE;
	RETURN;
END_IF

ptNvoLastInternalUse^.1 := FALSE;
ptNvoInternalUse^ := ptNvoLastInternalUse^;
FuMemCopy(ptNvo, ptNvoLast, uiNvoVariableLength);

FuDoNvoUpdate_Module_1 := TRUE;
END_FUNCTION

(* POU LON/Shared/Internal/FuSnvtFileStatusToRaw, ST *)
FUNCTION FuSnvtFileStatusToRaw : BOOL
(******************************************)
(* Automatic generated code, do not edit! *)
(******************************************)
VAR_INPUT
	NvDataIn :  POINTER TO typSnvtFileStatus;
	DataOut : POINTER TO ARRAY[0..26] OF BYTE;
END_VAR
VAR
END_VAR
DataOut^[0] := NvDataIn^.bStatus;

DataOut^[1] := WORD_TO_BYTE(SHR(NvDataIn^.wNumberOfFiles, 8));
DataOut^[2] := WORD_TO_BYTE(NvDataIn^.wNumberOfFiles);

DataOut^[3] := WORD_TO_BYTE(SHR(NvDataIn^.wSelectedFile, 8));
DataOut^[4] := WORD_TO_BYTE(NvDataIn^.wSelectedFile);

DataOut^[5] := NvDataIn^.abAdr[0];
DataOut^[6] := NvDataIn^.abAdr[1];
DataOut^[7] := NvDataIn^.abAdr[2];
DataOut^[8] := NvDataIn^.abAdr[3];
DataOut^[9] := NvDataIn^.abAdr[4];
DataOut^[10] := NvDataIn^.abAdr[5];
DataOut^[11] := NvDataIn^.abAdr[6];
DataOut^[12] := NvDataIn^.abAdr[7];
DataOut^[13] := NvDataIn^.abAdr[8];
DataOut^[14] := NvDataIn^.abAdr[9];
DataOut^[15] := NvDataIn^.abAdr[10];
DataOut^[16] := NvDataIn^.abAdr[11];
DataOut^[17] := NvDataIn^.abAdr[12];
DataOut^[18] := NvDataIn^.abAdr[13];
DataOut^[19] := NvDataIn^.abAdr[14];
DataOut^[20] := NvDataIn^.abAdr[15];
DataOut^[21] := NvDataIn^.abAdr[16];
DataOut^[22] := NvDataIn^.abAdr[17];
DataOut^[23] := NvDataIn^.abAdr[18];
DataOut^[24] := NvDataIn^.abAdr[19];
DataOut^[25] := NvDataIn^.abAdr[20];
DataOut^[26] := NvDataIn^.abAdr[21];

FuSnvtFileStatusToRaw := TRUE;
END_FUNCTION

(* POU LON/Module_1/Internal/FuSendNviValueReq_Module_1, ST *)
FUNCTION FuSendNviValueReq_Module_1 : BOOL
(******************************************)
(* Automatic generated code, do not edit! *)
(******************************************)
VAR_INPUT
	ptInternalUseOnly : POINTER TO BYTE;
	bNvIndex : BYTE;
END_VAR
IF ptInternalUseOnly^.0 = TRUE THEN
	OutDataTelegram_Module_1[0] := C2M_NV_VALUE_QRY;
	OutDataTelegram_Module_1[1] := bNvIndex;

	mbxModule_1.bTxPrio := 1;
	mbxModule_1.bTxProtID := 0;
	mbxModule_1.pbTxData := ADR(OutDataTelegram_Module_1);
	mbxModule_1.unTxLen := 2;
	mbxModule_1.MBX_SEND();

	IF (mbxModule_1.nError <> MBX_OK) THEN
		FuSendNviValueReq_Module_1 := FALSE;
		RETURN;
	END_IF
	ptInternalUseOnly^.0 := FALSE;
END_IF

FuSendNviValueReq_Module_1 := TRUE;
END_FUNCTION

(* POU LON/Module_1/NV_Interface/Module_1_Virtualfunctionalblock, ST *)
FUNCTION_BLOCK Module_1_Virtualfunctionalblock
(******************************************)
(* Automatic generated code, do not edit! *)
(******************************************)
VAR_INPUT
	bObjectIndex : BYTE := 0;
	VT_Request : typSnvtObjRequest;
	VT_TimeSet : typSnvtTimeStamp;
	VT_AlarmSet : typSnvtAlarm;
	VT_DHW_ModeSet : typSnvtHvacMode;
	VT_DHW_SetPoint : typSnvtTempP;
	VT_CFD_SetEnable : typSnvtSwitch;
	VT_CFD_SetMode : typSnvtHvacMode;
	VT_CFD_SetPoint : typSnvtTempP;

END_VAR
VAR_OUTPUT
	VT_Status : typSnvtObjStatus;
	VT_Alarm : typSnvtAlarm;
	VT_RlyState : typSnvtState;
	VT_DHW_ActTemp : typSnvtTempP;
	VT_DHW_SetTemp : typSnvtTempP;
	VT_CFD_GetEnable : typSnvtSwitch;
	VT_CFD_Temp : typSnvtTempP;
	VT_CFD_SetTemp : typSnvtTempP;

END_VAR
VAR
	xSetOnce : BOOL := TRUE;
	xDataInUpdated : BOOL := FALSE;
	VT_RequestLast: typSnvtObjRequest;
	VT_TimeSetLast: typSnvtTimeStamp;
	VT_AlarmSetLast: typSnvtAlarm;
	VT_CFD_SetEnableLast: typSnvtSwitch;
	paNviSnvtTempP : ARRAY[0..3] OF POINTER TO typSnvtTempP;
	aNviSnvtTempPIndex : ARRAY[0..3] OF BYTE := 7,9,13,15;
	paNvoSnvtHvacMode : ARRAY[0..1] OF POINTER TO typSnvtHvacMode;
	aNvoSnvtHvacModeIndex : ARRAY[0..1] OF BYTE := 6,12;
	aNvoSnvtHvacModeLast : ARRAY[0..1] OF typSnvtHvacMode;
	aNvoSnvtHvacModePriority : ARRAY[0..0] OF BYTE := 16#00;
	paNvoSnvtTempP : ARRAY[0..1] OF POINTER TO typSnvtTempP;
	aNvoSnvtTempPIndex : ARRAY[0..1] OF BYTE := 8,14;
	aNvoSnvtTempPLast : ARRAY[0..1] OF typSnvtTempP;
	aNvoSnvtTempPPriority : ARRAY[0..0] OF BYTE := 16#00;

	cmd : BYTE;
	z : INT;
	bNvRelativeIdx : BYTE;
	bNvAbsoluteIdx : BYTE;
	wCpRelativeIdx : WORD;
	wCpAbsoluteIdx : WORD;
END_VAR
VAR CONSTANT
	bNvStartIndex : BYTE := 5;
	wCpStartIndex : WORD := 65535;
	bLmoCount : BYTE := 1;
END_VAR
IF (xInitRunning_Module_1 = TRUE) AND (xSetOnce = TRUE) THEN
	xSetOnce := FALSE;
	CachePointers();
	SetUpdateFlags();
END_IF

CheckUpdateFlags();
IF (xInitRunning_Module_1 = FALSE) AND (xDataInUpdated = FALSE) THEN
	IF (mbxModule_1.bStatus.0) THEN
		SendValueRequest();
	END_IF
END_IF

IF (xInitRunning_Module_1 = FALSE) AND (mbxModule_1.bStatus.0) THEN
	xSetOnce := TRUE;
	xDataInUpdated := FALSE;
	IF ((NOT FuMemCompare(ADR(VT_RequestLast), ADR(VT_Request), ADR(VT_Request.bStatusInformation) - ADR(VT_Request))) OR (VT_Request.bStatusInformation.7 = TRUE) OR (VT_RequestLast.bInternalUseOnly.1 = TRUE)) THEN
		FuSnvtObjRequestToRaw(ADR(VT_Request), ADR(OutDataTelegram_Module_1[2]));

		bNvAbsoluteIdx := bNvStartIndex + bObjectIndex + (0 * bLmoCount);

		IF (FuDoNvoUpdate_Module_1(ADR(VT_Request), ADR(VT_RequestLast), ADR(VT_Request.bInternalUseOnly), ADR(VT_RequestLast.bInternalUseOnly), ADR(VT_Request.bStatusInformation), bNvAbsoluteIdx, 3, SIZEOF(VT_Request)) = FALSE) THEN
			RETURN;
		END_IF
	END_IF
	IF ((NOT FuMemCompare(ADR(VT_TimeSetLast), ADR(VT_TimeSet), ADR(VT_TimeSet.bStatusInformation) - ADR(VT_TimeSet))) OR (VT_TimeSet.bStatusInformation.7 = TRUE) OR (VT_TimeSetLast.bInternalUseOnly.1 = TRUE)) THEN
		FuSnvtTimeStampToRaw(ADR(VT_TimeSet), ADR(OutDataTelegram_Module_1[2]));

		bNvAbsoluteIdx := bNvStartIndex + bObjectIndex + (2 * bLmoCount);

		IF (FuDoNvoUpdate_Module_1(ADR(VT_TimeSet), ADR(VT_TimeSetLast), ADR(VT_TimeSet.bInternalUseOnly), ADR(VT_TimeSetLast.bInternalUseOnly), ADR(VT_TimeSet.bStatusInformation), bNvAbsoluteIdx, 7, SIZEOF(VT_TimeSet)) = FALSE) THEN
			RETURN;
		END_IF
	END_IF
	IF ((NOT FuMemCompare(ADR(VT_AlarmSetLast), ADR(VT_AlarmSet), ADR(VT_AlarmSet.bStatusInformation) - ADR(VT_AlarmSet))) OR (VT_AlarmSet.bStatusInformation.7 = TRUE) OR (VT_AlarmSetLast.bInternalUseOnly.1 = TRUE)) THEN
		FuSnvtAlarmToRaw(ADR(VT_AlarmSet), ADR(OutDataTelegram_Module_1[2]));

		bNvAbsoluteIdx := bNvStartIndex + bObjectIndex + (4 * bLmoCount);

		IF (FuDoNvoUpdate_Module_1(ADR(VT_AlarmSet), ADR(VT_AlarmSetLast), ADR(VT_AlarmSet.bInternalUseOnly), ADR(VT_AlarmSetLast.bInternalUseOnly), ADR(VT_AlarmSet.bStatusInformation), bNvAbsoluteIdx, 29, SIZEOF(VT_AlarmSet)) = FALSE) THEN
			RETURN;
		END_IF
	END_IF
	IF ((NOT FuMemCompare(ADR(VT_CFD_SetEnableLast), ADR(VT_CFD_SetEnable), ADR(VT_CFD_SetEnable.bStatusInformation) - ADR(VT_CFD_SetEnable))) OR (VT_CFD_SetEnable.bStatusInformation.7 = TRUE) OR (VT_CFD_SetEnableLast.bInternalUseOnly.1 = TRUE)) THEN
		FuSnvtSwitchToRaw(ADR(VT_CFD_SetEnable), ADR(OutDataTelegram_Module_1[2]));

		bNvAbsoluteIdx := bNvStartIndex + bObjectIndex + (10 * bLmoCount);

		IF (FuDoNvoUpdate_Module_1(ADR(VT_CFD_SetEnable), ADR(VT_CFD_SetEnableLast), ADR(VT_CFD_SetEnable.bInternalUseOnly), ADR(VT_CFD_SetEnableLast.bInternalUseOnly), ADR(VT_CFD_SetEnable.bStatusInformation), bNvAbsoluteIdx, 2, SIZEOF(VT_CFD_SetEnable)) = FALSE) THEN
			RETURN;
		END_IF
	END_IF
	FOR z := 0 TO 1 DO
		IF ((NOT FuMemCompare(ADR(aNvoSnvtHvacModeLast[z]), paNvoSnvtHvacMode[z], ADR(paNvoSnvtHvacMode[z]^.bStatusInformation) - paNvoSnvtHvacMode[z])) OR (paNvoSnvtHvacMode[z]^.bStatusInformation.7 = TRUE) OR (aNvoSnvtHvacModeLast[z].bInternalUseOnly.1 = TRUE)) THEN
			FuSnvtHvacModeToRaw(paNvoSnvtHvacMode[z], ADR(OutDataTelegram_Module_1[2]));

			bNvAbsoluteIdx := bNvStartIndex + bObjectIndex + (aNvoSnvtHvacModeIndex[z] * bLmoCount);

			IF (FuDoNvoUpdate_Module_1(paNvoSnvtHvacMode[z], ADR(aNvoSnvtHvacModeLast[z]), ADR(paNvoSnvtHvacMode[z]^.bInternalUseOnly), ADR(aNvoSnvtHvacModeLast[z].bInternalUseOnly), ADR(paNvoSnvtHvacMode[z]^.bStatusInformation), bNvAbsoluteIdx, 1, SIZEOF(aNvoSnvtHvacModeLast[z])) = FALSE) THEN
				RETURN;
			END_IF
		END_IF
	END_FOR
	FOR z := 0 TO 1 DO
		IF ((NOT FuMemCompare(ADR(aNvoSnvtTempPLast[z]), paNvoSnvtTempP[z], ADR(paNvoSnvtTempP[z]^.bStatusInformation) - paNvoSnvtTempP[z])) OR (paNvoSnvtTempP[z]^.bStatusInformation.7 = TRUE) OR (aNvoSnvtTempPLast[z].bInternalUseOnly.1 = TRUE)) THEN
			FuSnvtTempPToRaw(paNvoSnvtTempP[z], ADR(OutDataTelegram_Module_1[2]));

			bNvAbsoluteIdx := bNvStartIndex + bObjectIndex + (aNvoSnvtTempPIndex[z] * bLmoCount);

			IF (FuDoNvoUpdate_Module_1(paNvoSnvtTempP[z], ADR(aNvoSnvtTempPLast[z]), ADR(paNvoSnvtTempP[z]^.bInternalUseOnly), ADR(aNvoSnvtTempPLast[z].bInternalUseOnly), ADR(paNvoSnvtTempP[z]^.bStatusInformation), bNvAbsoluteIdx, 2, SIZEOF(aNvoSnvtTempPLast[z])) = FALSE) THEN
				RETURN;
			END_IF
		END_IF
	END_FOR

END_IF
END_FUNCTION_BLOCK
ACTION CachePointers:
paNviSnvtTempP[0] := ADR(VT_DHW_ActTemp);
paNviSnvtTempP[1] := ADR(VT_DHW_SetTemp);
paNviSnvtTempP[2] := ADR(VT_CFD_Temp);
paNviSnvtTempP[3] := ADR(VT_CFD_SetTemp);
paNvoSnvtHvacMode[0] := ADR(VT_DHW_ModeSet);
paNvoSnvtHvacMode[1] := ADR(VT_CFD_SetMode);
paNvoSnvtTempP[0] := ADR(VT_DHW_SetPoint);
paNvoSnvtTempP[1] := ADR(VT_CFD_SetPoint);
;
END_ACTION
ACTION CheckUpdateFlags:
xDataInUpdated := (NOT VT_Status.bInternalUseOnly.0) AND (NOT VT_Alarm.bInternalUseOnly.0) AND (NOT VT_RlyState.bInternalUseOnly.0) AND (NOT VT_CFD_GetEnable.bInternalUseOnly.0) AND TRUE;
FOR z := 0 TO 3 DO
	xDataInUpdated := xDataInUpdated AND (NOT paNviSnvtTempP[z]^.bInternalUseOnly.0);
END_FOR
END_ACTION
ACTION DataReceived:
cmd := InDataTelegram_Module_1[0];
IF (cmd = M2C_NVI_UPDT_OCCD) OR (cmd = M2C_NV_VALUE_RSP) OR (cmd = M2C_NVI_UPDT_TOUT) THEN
	bNvRelativeIdx := (InDataTelegram_Module_1[1] - bNvStartIndex - bObjectIndex) / bLmoCount;
	CASE bNvRelativeIdx OF
	1:
		IF (cmd = M2C_NVI_UPDT_OCCD) OR (cmd = M2C_NV_VALUE_RSP) THEN
			IF (unLastLen_mbxModule_1 = (2 + 6)) THEN
				FuRawToSnvtObjStatus(ADR(InDataTelegram_Module_1[2]), ADR(VT_Status));
				VT_Status.bInternalUseOnly.0 := FALSE;
				VT_Status.bStatusInformation := FuInkrementNviStatus(VT_Status.bStatusInformation);
			ELSIF (unLastLen_mbxModule_1 = 2) THEN
				VT_Status.bStatusInformation := FuInkrementNviStatus(VT_Status.bStatusInformation);
			END_IF
		ELSIF (cmd = M2C_NVI_UPDT_TOUT) THEN
			IF (unLastLen_mbxModule_1 = 3) THEN
				VT_Status.bStatusInformation.4 := BYTE_TO_BOOL(InDataTelegram_Module_1[2]);
			END_IF
		END_IF
	3:
		IF (cmd = M2C_NVI_UPDT_OCCD) OR (cmd = M2C_NV_VALUE_RSP) THEN
			IF (unLastLen_mbxModule_1 = (2 + 29)) THEN
				FuRawToSnvtAlarm(ADR(InDataTelegram_Module_1[2]), ADR(VT_Alarm));
				VT_Alarm.bInternalUseOnly.0 := FALSE;
				VT_Alarm.bStatusInformation := FuInkrementNviStatus(VT_Alarm.bStatusInformation);
			ELSIF (unLastLen_mbxModule_1 = 2) THEN
				VT_Alarm.bStatusInformation := FuInkrementNviStatus(VT_Alarm.bStatusInformation);
			END_IF
		ELSIF (cmd = M2C_NVI_UPDT_TOUT) THEN
			IF (unLastLen_mbxModule_1 = 3) THEN
				VT_Alarm.bStatusInformation.4 := BYTE_TO_BOOL(InDataTelegram_Module_1[2]);
			END_IF
		END_IF
	5:
		IF (cmd = M2C_NVI_UPDT_OCCD) OR (cmd = M2C_NV_VALUE_RSP) THEN
			IF (unLastLen_mbxModule_1 = (2 + 2)) THEN
				FuRawToSnvtState(ADR(InDataTelegram_Module_1[2]), ADR(VT_RlyState));
				VT_RlyState.bInternalUseOnly.0 := FALSE;
				VT_RlyState.bStatusInformation := FuInkrementNviStatus(VT_RlyState.bStatusInformation);
			ELSIF (unLastLen_mbxModule_1 = 2) THEN
				VT_RlyState.bStatusInformation := FuInkrementNviStatus(VT_RlyState.bStatusInformation);
			END_IF
		ELSIF (cmd = M2C_NVI_UPDT_TOUT) THEN
			IF (unLastLen_mbxModule_1 = 3) THEN
				VT_RlyState.bStatusInformation.4 := BYTE_TO_BOOL(InDataTelegram_Module_1[2]);
			END_IF
		END_IF
	11:
		IF (cmd = M2C_NVI_UPDT_OCCD) OR (cmd = M2C_NV_VALUE_RSP) THEN
			IF (unLastLen_mbxModule_1 = (2 + 2)) THEN
				FuRawToSnvtSwitch(ADR(InDataTelegram_Module_1[2]), ADR(VT_CFD_GetEnable));
				VT_CFD_GetEnable.bInternalUseOnly.0 := FALSE;
				VT_CFD_GetEnable.bStatusInformation := FuInkrementNviStatus(VT_CFD_GetEnable.bStatusInformation);
			ELSIF (unLastLen_mbxModule_1 = 2) THEN
				VT_CFD_GetEnable.bStatusInformation := FuInkrementNviStatus(VT_CFD_GetEnable.bStatusInformation);
			END_IF
		ELSIF (cmd = M2C_NVI_UPDT_TOUT) THEN
			IF (unLastLen_mbxModule_1 = 3) THEN
				VT_CFD_GetEnable.bStatusInformation.4 := BYTE_TO_BOOL(InDataTelegram_Module_1[2]);
			END_IF
		END_IF
	7, 9, 13, 15:
		IF (cmd = M2C_NVI_UPDT_OCCD) OR (cmd = M2C_NV_VALUE_RSP) THEN
			IF (unLastLen_mbxModule_1 = (2 + 2)) THEN
				FOR z := 0 TO 3 DO
					IF aNviSnvtTempPIndex[z] = bNvRelativeIdx THEN
						FuRawToSnvtTempP(ADR(InDataTelegram_Module_1[2]), paNviSnvtTempP[z]);
						paNviSnvtTempP[z]^.bInternalUseOnly.0 := FALSE;
						paNviSnvtTempP[z]^.bStatusInformation := FuInkrementNviStatus(paNviSnvtTempP[z]^.bStatusInformation);
						EXIT;
					END_IF
				END_FOR
			ELSIF (unLastLen_mbxModule_1 = 2) THEN
				FOR z := 0 TO 3 DO
					IF aNviSnvtTempPIndex[z] = bNvRelativeIdx THEN
						paNviSnvtTempP[z]^.bStatusInformation := FuInkrementNviStatus(paNviSnvtTempP[z]^.bStatusInformation);
						EXIT;
					END_IF
				END_FOR
			END_IF
		ELSIF (cmd = M2C_NVI_UPDT_TOUT) THEN
			IF (unLastLen_mbxModule_1 = 3) THEN
				FOR z := 0 TO 3 DO
					IF aNviSnvtTempPIndex[z] = bNvRelativeIdx THEN
						paNviSnvtTempP[z]^.bStatusInformation.4 := BYTE_TO_BOOL(InDataTelegram_Module_1[2]);
						EXIT;
					END_IF
				END_FOR
			END_IF
		END_IF

	END_CASE
ELSIF (cmd = M2C_CP_VALUE_RSP) THEN
	wCpRelativeIdx := ((InDataTelegram_Module_1[1] + InDataTelegram_Module_1[2] * 256) - wCpStartIndex - bObjectIndex) / bLmoCount;
	CASE wCpRelativeIdx OF

	END_CASE
END_IF
END_ACTION
ACTION ResetNviUpdate:
VT_Status.bStatusInformation := VT_Status.bStatusInformation AND 16#F8;
VT_Alarm.bStatusInformation := VT_Alarm.bStatusInformation AND 16#F8;
VT_RlyState.bStatusInformation := VT_RlyState.bStatusInformation AND 16#F8;
VT_CFD_GetEnable.bStatusInformation := VT_CFD_GetEnable.bStatusInformation AND 16#F8;
FOR z := 0 TO 3 DO
	paNviSnvtTempP[z]^.bStatusInformation := paNviSnvtTempP[z]^.bStatusInformation AND 16#F8;
END_FOR
;
END_ACTION
ACTION SendValueRequest:
IF (FuSendNviValueReq_Module_1(ADR(VT_Status.bInternalUseOnly), bNvStartIndex + bObjectIndex + (1 * bLmoCount)) = FALSE) THEN
	RETURN;
END_IF

IF (FuSendNviValueReq_Module_1(ADR(VT_Alarm.bInternalUseOnly), bNvStartIndex + bObjectIndex + (3 * bLmoCount)) = FALSE) THEN
	RETURN;
END_IF

IF (FuSendNviValueReq_Module_1(ADR(VT_RlyState.bInternalUseOnly), bNvStartIndex + bObjectIndex + (5 * bLmoCount)) = FALSE) THEN
	RETURN;
END_IF

IF (FuSendNviValueReq_Module_1(ADR(VT_CFD_GetEnable.bInternalUseOnly), bNvStartIndex + bObjectIndex + (11 * bLmoCount)) = FALSE) THEN
	RETURN;
END_IF

FOR z := 0 TO 3 DO
	IF (FuSendNviValueReq_Module_1(ADR(paNviSnvtTempP[z]^.bInternalUseOnly), bNvStartIndex + bObjectIndex + (aNviSnvtTempPIndex[z] * bLmoCount)) = FALSE) THEN
		RETURN;
	END_IF;
END_FOR;
;
END_ACTION
ACTION SetUpdateFlags:
VT_RequestLast.bInternaluseOnly.1 := TRUE;
VT_RequestLast.bInternaluseOnly.7 := FALSE;
VT_Status.bInternaluseOnly.0 := TRUE;
VT_TimeSetLast.bInternaluseOnly.1 := TRUE;
VT_TimeSetLast.bInternaluseOnly.7 := FALSE;
VT_Alarm.bInternaluseOnly.0 := TRUE;
VT_AlarmSetLast.bInternaluseOnly.1 := TRUE;
VT_AlarmSetLast.bInternaluseOnly.7 := FALSE;
VT_RlyState.bInternaluseOnly.0 := TRUE;
VT_CFD_SetEnableLast.bInternaluseOnly.1 := TRUE;
VT_CFD_SetEnableLast.bInternaluseOnly.7 := FALSE;
VT_CFD_GetEnable.bInternaluseOnly.0 := TRUE;
FOR z := 0 TO 3 DO
	paNviSnvtTempP[z]^.bInternaluseOnly.0 := TRUE;
END_FOR;
FOR z := 0 TO 1 DO
	aNvoSnvtHvacModeLast[z].bInternaluseOnly.1 := TRUE;
	aNvoSnvtHvacModeLast[z].bInternaluseOnly.7 := (SHR(aNvoSnvtHvacModePriority[z / 8], z MOD 8) AND 1) <> 0;
END_FOR;
FOR z := 0 TO 1 DO
	aNvoSnvtTempPLast[z].bInternaluseOnly.1 := TRUE;
	aNvoSnvtTempPLast[z].bInternaluseOnly.7 := (SHR(aNvoSnvtTempPPriority[z / 8], z MOD 8) AND 1) <> 0;
END_FOR;
;
END_ACTION

(* POU LON/Shared/Internal/FuSnvtObjRequestToRaw, ST *)
FUNCTION FuSnvtObjRequestToRaw : BOOL
(******************************************)
(* Automatic generated code, do not edit! *)
(******************************************)
VAR_INPUT
	NvDataIn :  POINTER TO typSnvtObjRequest;
	DataOut : POINTER TO ARRAY[0..2] OF BYTE;
END_VAR
VAR
END_VAR
DataOut^[0] := WORD_TO_BYTE(SHR(NvDataIn^.wObjectId, 8));
DataOut^[1] := WORD_TO_BYTE(NvDataIn^.wObjectId);

DataOut^[2] := NvDataIn^.bObjectRequest;

FuSnvtObjRequestToRaw := TRUE;
END_FUNCTION

(* POU LON/Shared/Internal/FuSnvtTimeStampToRaw, ST *)
FUNCTION FuSnvtTimeStampToRaw : BOOL
(******************************************)
(* Automatic generated code, do not edit! *)
(******************************************)
VAR_INPUT
	NvDataIn :  POINTER TO typSnvtTimeStamp;
	DataOut : POINTER TO ARRAY[0..6] OF BYTE;
END_VAR
VAR
END_VAR
DataOut^[0] := INT_TO_BYTE(SHR(NvDataIn^.iYear, 8));
DataOut^[1] := INT_TO_BYTE(NvDataIn^.iYear);

DataOut^[2] := NvDataIn^.bMonth;

DataOut^[3] := NvDataIn^.bDay;

DataOut^[4] := NvDataIn^.bHour;

DataOut^[5] := NvDataIn^.bMinute;

DataOut^[6] := NvDataIn^.bSecond;

FuSnvtTimeStampToRaw := TRUE;
END_FUNCTION

(* POU LON/Shared/Internal/FuSnvtAlarmToRaw, ST *)
FUNCTION FuSnvtAlarmToRaw : BOOL
(******************************************)
(* Automatic generated code, do not edit! *)
(******************************************)
VAR_INPUT
	NvDataIn :  POINTER TO typSnvtAlarm;
	DataOut : POINTER TO ARRAY[0..28] OF BYTE;
END_VAR
VAR
END_VAR
DataOut^[0] := NvDataIn^.abLocation[0];
DataOut^[1] := NvDataIn^.abLocation[1];
DataOut^[2] := NvDataIn^.abLocation[2];
DataOut^[3] := NvDataIn^.abLocation[3];
DataOut^[4] := NvDataIn^.abLocation[4];
DataOut^[5] := NvDataIn^.abLocation[5];

DataOut^[6] := WORD_TO_BYTE(SHR(NvDataIn^.wObjectId, 8));
DataOut^[7] := WORD_TO_BYTE(NvDataIn^.wObjectId);

DataOut^[8] := NvDataIn^.bAlarmType;

DataOut^[9] := NvDataIn^.bPriorityLevel;

DataOut^[10] := WORD_TO_BYTE(SHR(NvDataIn^.wIndexToSnvt, 8));
DataOut^[11] := WORD_TO_BYTE(NvDataIn^.wIndexToSnvt);

DataOut^[12] := NvDataIn^.abValue[0];
DataOut^[13] := NvDataIn^.abValue[1];
DataOut^[14] := NvDataIn^.abValue[2];
DataOut^[15] := NvDataIn^.abValue[3];

DataOut^[16] := WORD_TO_BYTE(SHR(NvDataIn^.wYear, 8));
DataOut^[17] := WORD_TO_BYTE(NvDataIn^.wYear);

DataOut^[18] := NvDataIn^.bMonth;

DataOut^[19] := NvDataIn^.bDay;

DataOut^[20] := NvDataIn^.bHour;

DataOut^[21] := NvDataIn^.bMinute;

DataOut^[22] := NvDataIn^.bSecond;

DataOut^[23] := WORD_TO_BYTE(SHR(NvDataIn^.wMillisecond, 8));
DataOut^[24] := WORD_TO_BYTE(NvDataIn^.wMillisecond);

DataOut^[25] := NvDataIn^.abAlarmLimit[0];
DataOut^[26] := NvDataIn^.abAlarmLimit[1];
DataOut^[27] := NvDataIn^.abAlarmLimit[2];
DataOut^[28] := NvDataIn^.abAlarmLimit[3];

FuSnvtAlarmToRaw := TRUE;
END_FUNCTION

(* POU LON/Shared/Internal/FuSnvtSwitchToRaw, ST *)
FUNCTION FuSnvtSwitchToRaw : BOOL
(******************************************)
(* Automatic generated code, do not edit! *)
(******************************************)
VAR_INPUT
	NvDataIn :  POINTER TO typSnvtSwitch;
	DataOut : POINTER TO ARRAY[0..1] OF BYTE;
END_VAR
VAR
END_VAR
DataOut^[0] := NvDataIn^.bValue;

DataOut^[1] := NvDataIn^.siState;

FuSnvtSwitchToRaw := TRUE;
END_FUNCTION

(* POU LON/Shared/Internal/FuSnvtHvacModeToRaw, ST *)
FUNCTION FuSnvtHvacModeToRaw : BOOL
(******************************************)
(* Automatic generated code, do not edit! *)
(******************************************)
VAR_INPUT
	NvDataIn :  POINTER TO typSnvtHvacMode;
	DataOut : POINTER TO ARRAY[0..0] OF BYTE;
END_VAR
VAR
END_VAR
DataOut^[0] := NvDataIn^.bSnvtHvacMode;

FuSnvtHvacModeToRaw := TRUE;
END_FUNCTION

(* POU LON/Shared/Internal/FuSnvtTempPToRaw, ST *)
FUNCTION FuSnvtTempPToRaw : BOOL
(******************************************)
(* Automatic generated code, do not edit! *)
(******************************************)
VAR_INPUT
	NvDataIn :  POINTER TO typSnvtTempP;
	DataOut : POINTER TO ARRAY[0..1] OF BYTE;
END_VAR
VAR
END_VAR
DataOut^[0] := INT_TO_BYTE(SHR(NvDataIn^.iSnvtTempP, 8));
DataOut^[1] := INT_TO_BYTE(NvDataIn^.iSnvtTempP);

FuSnvtTempPToRaw := TRUE;
END_FUNCTION

(* POU TCP_Logger/Logger_Proc, ST *)
PROGRAM Logger_Proc
VAR
	c1:         	TCPCLIENT;

	Open:	    	BOOL;
	IpAddr:			DWORD;
	InetAddr:		DWORD;
	Connected:  	BOOL;
	Error:      	DINT;
	TxTrig:     	BOOL;
	RxData:			ARRAY [0..MAX_RECEIVE_TCP_CLIENT] OF BYTE;
	RxLen:			DINT;

	Retry:			BYTE;	(* Counter for connection retries *)
	Recovered:		BYTE;	(* Counter for recovered unsent messages *)

	i:				DINT;
	pos:			DWORD;
	hFile:			DWORD;

END_VAR
(*=== State machine ===*)
CASE Logger.Status OF

	S_Logger_UNKNOWN:
		(* Startup *)
		Logger.SendReq:=FALSE;
		Open:=FALSE;
		Logger.Status:=S_Logger_IDLE;

	S_Logger_IDLE:
		(* Wait request *)
		IF Logger.SendReq THEN
			(* Resolve server name or use static IP *)
			IF LEN(Logger_SERVER)=0 THEN
				InetAddr:=SysSockInetAddr(Logger_IP);
			ELSE
				IpAddr:=SysSockGetHostByName(ADR(Logger_SERVER));
				DWORDSWAP(pIn:=ADR(IpAddr), pOut:=ADR(InetAddr));
			END_IF
			TxTrig:=FALSE;
			RxLen:=0;
			(* Open connection *)
			Open:=TRUE;
			Logger.Status:=S_Logger_WAITCONN;
		END_IF

	S_Logger_WAITCONN:
		(* Wait connection *)
		IF Connected THEN
			(* Send data *)
			TxTrig:=TRUE;
			Logger.Status:=S_Logger_WAITTX;
		END_IF
		IF Error>0 THEN
			Open:=FALSE;
			Logger.Status:=S_Logger_ERROR;
		END_IF

	S_Logger_WAITTX:
		(* Wait transmission *)
		IF NOT TxTrig THEN
			Logger.Status:=S_Logger_WAITRESP;
		END_IF
		IF Error>0 THEN
			Open:=FALSE;
			Logger.Status:=S_Logger_ERROR;
		END_IF

	S_Logger_WAITRESP:
		(* Wait response *)
		IF Connected=FALSE (* OR TIMEOUT!! *) THEN
			Open:=FALSE;
			(* Check response *)
			IF RxLen>=4 AND CHKSTRING(pString:=ADR(RxData), pPattern:=ADR(Logger_CHECK)) THEN
				Logger.SendReq:=FALSE;
				Retry:=0;
				(* Check unsent messages to flush *)
				IF Recovered<Logger_RecoverMsgs THEN
					MsgChk();
					IF Logger.SendReq=TRUE THEN
						Recovered:=Recovered+1;
					ELSE
						Recovered:=0;
					END_IF
				ELSE
					Recovered:=0;
				END_IF
				Logger.Status:=S_Logger_IDLE;
			ELSE
				Logger.Status:=S_Logger_ERROR;
			END_IF
		END_IF

	S_Logger_ERROR:
		(* Connection error or send failure *)
		Retry:=Retry+1;
		IF Retry>Logger_ConnRetries THEN
			(* Save message as unsent *)
			MsgSave();
			Logger.SendReq:=FALSE;
			Retry:=0;
		END_IF
		Logger.Status:=S_Logger_IDLE;

ELSE
	Logger.Status:=S_Logger_UNKNOWN;
END_CASE


(*=== Execute client lib ===*)
c1(
	xOpenConnection			:= Open,
	dwInetAddr 				:= InetAddr,
	wPortNumber				:= Logger_PORT,
	ptSendData				:= ADR(Logger.SendData),
	diSendCount				:= Logger.SendLen,
	tConnectWatchdogTime	:= t#10s,
	xStartSend				:= TxTrig,
	aReceiveBuffer			:= RxData,
	diReceiveCount			:= RxLen,
	xConnected				=> Connected,
	diError					=> Error
);

(*=== Process Rx data ===*)
(*IF RxLen>0 THEN
	RxLen:=0;
END_IF*)
END_PROGRAM
ACTION MsgChk:
(* Open index file *)
hFile:=SysFileOpen(Logger_IndexFile,'r');
IF hFile=0 THEN
	RETURN;
END_IF
(* Search oldest message to recover *)
SysFileSetPos(hFile,Logger.LastIdxPos);
Logger.SendLen:=0;
REPEAT
	SysFileRead(hFile, ADR(Logger.SendIdx), SIZEOF(Logger.SendIdx));
	pos:=SysFileGetPos(hFile);
	SysFileRead(hFile, ADR(Logger.SendLen), SIZEOF(Logger.SendLen));
UNTIL
	SysFileEOF(hFile) OR Logger.SendLen<>0
END_REPEAT
SysFileClose(hFile);
(* Delete index file when all messages are recovered *)
IF Logger.SendLen=0 THEN
	Logger.LastIdxPos:=0;
	SysFileDelete(Logger_IndexFile);
	RETURN;
END_IF
(* Recover message data *)
hFile:=SysFileOpen(Logger_DataFile,'r');
IF hFile<>0 THEN
	SysFileSetPos(hFile,Logger.SendIdx);
	SysFileRead(hFile,ADR(Logger.SendData),Logger.SendLen);
	Logger.SendReq:=TRUE;
	SysFileClose(hFile);
END_IF
(* Clear index entry *)
hFile:=SysFileOpen(Logger_IndexFile,'a');
IF hFile<>0 THEN
	SysFileSetPos(hFile,pos);
	i:=0;
	SysFileWrite(hFile, ADR(i), 4);
	Logger.LastIdxPos:=SysFileGetPos(hFile);
	SysFileClose(hFile);
END_IF
END_ACTION
ACTION MsgSave:
(* Add log position in recovery indexes *)
hFile:=SysFileOpen(Logger_IndexFile,'a');
SysFileWrite(hFile, ADR(Logger.SendIdx), SIZEOF(Logger.SendIdx));
SysFileWrite(hFile, ADR(Logger.SendLen), SIZEOF(Logger.SendLen));
SysFileClose(hFile);
END_ACTION

(* POU Utils Functions/TCPCLIENT, ST *)
FUNCTION_BLOCK TCPCLIENT
(***********************************************************************************************************	*)
(* Version: 1.3b                        			          													*)
(* Date: 28.10.2014                   				          							            			*)
(***********************************************************************************************************	*)
(* WAGO Kontakttechnik GmbH Hansastr. 27 32423 Minden(Westf.)													*)
(* Tel. +0049 571/887-0 Fax. +0049 571/887-0																	*)
(* Author: VB																									*)
(***********************************************************************************************************	*)
(*Description:	A TCP client to read and write data with additional connection watchdog							*)
(*History:																										*)
(*Version 1.3b: 28.10.2014: Use DWORD address for IP (Andrea Ravasio)											*)
(*Version 1.3: 11.02.2011: Changes according to 750-880/881											 			*)
(*Version 1.2: 29.08.2007 Bugfix TCP Client																		*)
(*Version 1.1: 15.01.2007 Changes according to FW11																*)
(*Version 1.0: 09.03.2006 Release																				*)
(***********************************************************************************************************	*)
VAR CONSTANT
	STATE_CREATE     				 : BYTE:= 0;
	STATE_OPEN     					 : BYTE:= 1;
	STATE_IOCTL    					 : BYTE:= 2;
	STATE_CONNECT     				 : BYTE:= 10;
	STATE_TX       					 : BYTE:= 20;
	STATE_RX       					 : BYTE:= 30;
	STATE_CLOSE    					 : BYTE:= 40;
	STATE_ERROR_TRAP			     : BYTE:= 200;
END_VAR

VAR_INPUT
	xOpenConnection					: BOOL;
	dwInetAddr						: DWORD; (* <== Use SysSockInetAddr() value or
													swapped bytes order of SysSockGetHostByName() value *)
	wPortNumber						: WORD;
	ptSendData						: POINTER TO ARRAY[0..MAX_SEND_TCP_CLIENT] OF BYTE;
	diSendCount						: DINT;
	tConnectWatchdogTime		    : TIME := t#10s;
END_VAR
VAR_OUTPUT
	xConnected						: BOOL;
	diError 						: DINT := 0;
END_VAR
(* ErrorCodes -----------------------------------------
	16#8001 => No socket descriptor available 
	16#8002 => SysSockSend returns -1 
	16#8003 => Socket was "gracefully closed" 
	16#8004 => switching to none blocking mode fails
	16#8005 => SysSockClose() returns FALSE 
    16#8006 => SysSockConnect() fails
    16#8007 => SysSockSend() fails
	16#8008 => error state machine 
	16#8009 => timeout while waiting for data from server 
------------------------------------------------------------*)
VAR_IN_OUT
	xStartSend							: BOOL;
	aReceiveBuffer						: ARRAY [0..MAX_RECEIVE_TCP_CLIENT] OF BYTE;
	diReceiveCount						: DINT;
END_VAR
VAR
	m_State								: BYTE := 0;
	m_ReceiveBuffer						: ARRAY [0..MAX_RECEIVE_TCP_CLIENT_SOCKET] OF BYTE;
	m_Socket							: DINT;
	m_AddressInfo						: SOCKADDRESS;
	m_BytesReceived						: DINT;
	m_diReturn							: DINT;
	m_xReturn							: BOOL;
	m_IoCtlParameter  					: DINT := 1; (* IOCTL-Parameter for non-blocking mode of sockets *)
	i									: INT;
	T_Connect							: TON;
	m_count								: DINT;
	diOption							: DINT := 1;
	m_Blocking   						: DINT := 0;
END_VAR
IF xOpenConnection THEN
	(* State maschine *)
	CASE  m_State OF

	(* -------------------------------------------------------------------------*)
	STATE_CREATE:
			(* create socket descriptor*)
			m_Socket := SysSockCreate(diAddressFamily	:= SOCKET_AF_INET,
													 diType		:= SOCKET_STREAM,
													 diProtocol := SOCKET_IPPROTO_TCP);
			IF m_Socket >= 0 THEN
			(*Set Push-Bit*)
				IF ADR(%MW0)=16#30000000  OR ADR(%MW0)=16#20000000 THEN (*841 or 881*)
					SysSockSetOption(
						diSocket:=m_Socket,
						diLevel:=6,
						diOption:=SOCKET_TCP_NODELAY,
						pOptionValue:=ADR(diOption),
						diOptionLength:=SIZEOF(diOption));
				ELSE
						;
				END_IF
				m_State := STATE_IOCTL; (* succesful *)
			ELSE
				diError := 16#8001;  (* no socket descriptor available *)
				m_State := STATE_ERROR_TRAP;
			END_IF

	(* -------------------------------------------------------------------------*)
	STATE_IOCTL: (* change  socket mode  to none blocking *)
		m_diReturn := SysSockIoctl( m_Socket, SOCKET_FIONBIO, ADR(m_IoCtlParameter));
		IF m_diReturn <> 0 THEN
			m_AddressInfo.sin_family := SOCKET_AF_INET;
			m_AddressInfo.sin_port := SysSockNtohs(wPortNumber);
			m_AddressInfo.sin_addr := dwInetAddr;
			m_State := STATE_CONNECT;
		ELSE
			diError := 16#8004;  (* switching to none blocking mode fails *)
			m_State := STATE_ERROR_TRAP;
		END_IF


	(* -------------------------------------------------------------------------*)
	STATE_CONNECT: (* connect with server *)
		T_Connect(IN:=TRUE , PT:=tConnectWatchdogTime);(*activate watchdog for establishing connection to a server*)
		m_xReturn := SysSockConnect ( m_Socket, ADR(m_AddressInfo),  SIZEOF(m_AddressInfo));
		IF m_xReturn THEN (* succesful *)
			IF xStartSend THEN
				m_State := STATE_TX;(*transmit data*)
			ELSE
				m_State := STATE_RX;(*wait for data from server*)
			END_IF
			xConnected:=TRUE;
			T_Connect(IN:=FALSE);
		ELSE
			IF T_Connect.Q THEN
				diError := 16#8006;  (* connect fails *)
				xConnected:=FALSE;
				T_Connect(IN:=FALSE);
				m_State := STATE_ERROR_TRAP;
				SysSockClose( m_Socket);
			ELSE
				m_State := STATE_CONNECT;(*client still  tries to set up connection*)
			END_IF
		END_IF


	STATE_TX:	 (* send TCP-message *)
		m_diReturn := SysSockSend(diSocket := m_Socket,
								  pbyBuffer := ADR(ptSendData^[0]),
								  diBufferSize := diSendCount-m_count,
								  diFlags := 0);

		CASE m_diReturn OF
		-1:	(* ERROR *)
			T_Connect(IN:=TRUE , PT:=CONNECT_WATCHDOG_TIME);(*activate watchdog to check communication*)
			IF t_Connect.Q THEN
				diError := 16#8007;
				T_Connect(IN:=FALSE);
				m_State:=STATE_CLOSE;
			END_IF
		0: (* socket was "gracefully closed" *)
			m_State := STATE_CLOSE;
			diError := 16#8003;
		ELSE (* succesful *)
			m_count:=m_count+m_diReturn;
			IF m_count>=diSendCount THEN
				diError := 16#0000;
				m_State := STATE_RX;
				m_count:=0;
				xStartSend:=FALSE;
			END_IF
			T_Connect(IN:=FALSE);
		END_CASE

	(* -------------------------------------------------------------------------*)
	STATE_RX: (* process receive data *)
			m_BytesReceived := SysSockRecv(	diSocket 	:= m_Socket,
										pbyBuffer 	:= ADR(m_ReceiveBuffer),		(* Address of receive buffer *)
										diBufferSize:= SIZEOF(m_ReceiveBuffer),
										diFlags		:= 0);

			CASE m_BytesReceived OF
			-1:	(* No data available or error occured *)
				T_Connect(IN:=TRUE , PT:=tConnectWatchdogTime);(*activate watchdog to check communication*)
				IF t_Connect.Q THEN
					diError:=16#8009;
					T_Connect(IN:=FALSE);
					m_State:=STATE_CLOSE;
				END_IF
				IF xStartSend THEN
					m_State:=STATE_TX	;(* WAIT IN THIS STATE  and check for arriving data or new send command*)
				END_IF;
			0: (* socket was "gracefully closed"  *)
				m_State:=STATE_CLOSE;
				diError := 16#8003;
			ELSE (* succesful *)
				diError := 16#0000;
				T_Connect(IN:=FALSE);
				(* Copy received data into receive buffer *)
				FOR i:= 0 TO DINT_TO_INT(m_BytesReceived	)-1 DO
					aReceiveBuffer[diReceiveCount]:= m_ReceiveBuffer[i];
					diReceiveCount:=(diReceiveCount+1) MOD SIZEOF(aReceiveBuffer);
				END_FOR

			END_CASE

